FUNCTION_BLOCK "SSA_SIEMENS_MICROMASTER"	// FB 1813
TITLE = SIEMENS MICROMASTER
//COPYRIGHT:    (C) 2004  BUHLER AG, CH-9240 UZWIL, SWITZERLAND
//
//PRODUCT:      SSA
//
//TITLE:        SIEMENS MICROMASTER Frequency Inverter Profibus Communication
//
//--------------------------------------------------------------------------------
//
//IDENT:         AUTHOR:             DEPT:                            DATE:
//
//FB1813.2.0     M.Wedler            AEB41                            25-Okt-2007
//               2nd Release
//FB1811.1.0     A.Egli              CT3                              13-Jul-2007
//               1st Release
//
//--------------------------------------------------------------------------------
//
//PURPOSE: 
//
//MANUAL : 
//
//RESTRICTIONS: 
//
//--------------------------------------------------------------------------------
//
AUTHOR : MW
FAMILY : STD
VERSION : 0.0
VAR
  InValuePC : INT ;	//Aktuel value 1 in [0.01 %]
  InEnableRev : BOOL ;
  InEnableFwd : BOOL ;
  CmdFaultReset : BOOL ;
  OutRunningRev : BOOL ;	//Feedback for element motor
  OutRunningFwd : BOOL ;	//Feedback for element motor
  OutFault : BOOL ;	//Feedback for element motor
  MotorStStopped : BOOL ;	//Motor has come to a standstill after stopping time
  Spare : BOOL ;
  OutValuePC : INT ;	//Setpoint value 1 in [0.01 %]
  Input : STRUCT
   StateWord_1 : STRUCT 	//Statuswort MICROMASTER
    DREHZAHL_ABWEICHUNG_OK : BOOL ;	//0=Nicht im Toleranzband             1=Soll-Ist-Überwachung im Toleranzband
    FUEHRUNG : BOOL ;	//0=Fuehrung Lokal                    1=Fuehrung SPS
    VERGLEICHSWERT : BOOL ;	//0=Vergleichswert nicht erreicht     1=Vergleichswert erreicht/ueberschritten
    GRENZE_ERREICHT : BOOL ;	//0=I-, M- oder P-Grenze erreicht     1=I-, M- oder P-Grenze nicht erreicht
    HALTEBREMSE : BOOL ;	//0=Motor Haltebremse                 1=Steuern Haltebremse
    WARN_UEBERTEMP_MOTOR : BOOL ;	//0=Warnung nicht wirksam             1=Warnung Übertemperatur Motor wirksam
    DREH_RECHTS : BOOL ;	//0=Linkslauf                         1=Rechtslauf
    WARNUNG_UEBERTEMP_FU : BOOL ;	//0=Warnung thermische Überlast Umrichter 1=Keine Warnung wirksam
    EINSCHALTBEREIT : BOOL ;	//0=Nicht einschaltbereit             1=Einschaltbereit
    BETRIEBSBEREIT : BOOL ;	//0=Nicht betriebsbereit              1=Betriebsbereit
    BETRIEB_FREIGEGEBEN : BOOL ;	//0=Betrieb gesperrt   1=Betrieb freigegeben->Hochlauf auf anliegendem Sollwert
    STOERUNG : BOOL ;	//0=Keine Störung wirksam             1=Störung wirksam
    AUS_2 : BOOL ;	//0=Austrudeln aktiv (AUS2)           1=Kein AUS2 aktiv
    AUS_3 : BOOL ;	//0=Schnellhalt aktiv (AUS3)          1=Kein AUS3 aktiv
    EINSCHALTSPERRE : BOOL ;	//1=Einschaltsperre -> Wiedereinschalten durch AUS1 und anschließendes EIN
    WARNUNG : BOOL ;	//0=Keine Warnung wirksam             1=Warnung wirksam, Motor weiter im Betrieb
   END_STRUCT ;
   ActualValue01 : INT ;	//Hauptistwert / Prozessdaten PD2
   ActualValue02 : INT ;	//Prozessdaten PD3
   ActualValue03 : INT ;	//Prozessdaten PD4
   ActualValue04 : INT ;	//Prozessdaten PD5
   ActualValue05 : INT ;	//Prozessdaten PD6
  END_STRUCT ;
  Output : STRUCT
   ControlWord_1 : STRUCT 	//Steuerwort MICROMASTER
    TIPPEN_RECHTS : BOOL ;	//1=Tippen rechts
    TIPPEN_LINKS : BOOL ;	//1=Tippen links
    PZD_GUELTIG : BOOL ;	//0=Sollwerte ungueltig              1=Sollwerte gueltig
    DREHRICHTUNGSUMKEHR : BOOL ;	//Drehrichtungsumkehr: 0=Rechtsdrehfeld / 1=Linksdrehfeld
    CONTROL_WORD_BIT_12 : BOOL ;	//reserviert
    MOTOR_POTI_HIGH : BOOL ;	//1=Motorpotentiometer höher
    MOTOR_POTI_DOWN : BOOL ;	//1=Motorpotentiometer tiefer
    LOCAL : BOOL ;	//0=Fern-Steuerung aktiv             1=Vorort-Steuerung aktiv
    AUS1 : BOOL ;	//0=AUS1->Abbremsen an der Rücklauframpe   1=EIN
    AUS2 : BOOL ;	//0=Austrudeln (AUS2)                      1=kein Austrudeln
    AUS3 : BOOL ;	//0=Schnellhalt (AUS3)->Abbremsen an der Schnellhalt-Rampe  1=kein Schnellhalt
    BETRIEB_FREIGEBEN : BOOL ;	//0=Betrieb sperren        1=Betrieb freigeben->Hochlauf mit anliegendem Sollwert
    HOCHLAUF_SPERREN : BOOL ;	//0=Hochlaufgeber wird auf NULL gesetzt    1=Hochlaufgeber freigeben
    HOCHLAUF_STOPPEN : BOOL ;	//0=Hochlaufgeber einfrieren               1=Hochlaufgeber freigeben
    SOLLWERT_FREIGEBEN : BOOL ;	//0=Drehzahlsollwert wird auf NULL gesetzt 1=Drehzahlsollwert freigeben
    FEHLER_QUITTIEREN : BOOL ;	//Flanke 0 -> 1 = Fehler quittieren, quittiert alle aktuellen Störungen
   END_STRUCT ;
   SetpointValue01 : INT ;	//Hauptsollwert / Prozessdaten PD2
   SetpointValue02 : INT ;	//Prozessdaten PD3
   SetpointValue03 : INT ;	//Prozessdaten PD4
   SetpointValue04 : INT ;	//Prozessdaten PD5
   SetpointValue05 : INT ;	//Prozessdaten PD6
  END_STRUCT ;
  Par : STRUCT
   spare1 : INT ;
   spare2 : INT ;
   spare3 : INT ;
   ParMovidrive : BOOL ;
   ParSinamics : BOOL ;
   ParMicromaster : BOOL ;
   ParABB : BOOL ;
   ParNord : BOOL ;
   ParDanfoss : BOOL ;
   ParIOByteNo : INT ;
  END_STRUCT ;
END_VAR
VAR_TEMP
  tmpAddrDB : INT ;
  tmpAddrIO : DINT ;
  tmpAddrInputFU : DINT ;
  tmpAddrOutputFU : DINT ;
END_VAR
BEGIN
NETWORK
TITLE = Calculate Address of Inverter
      L     #Par.ParIOByteNo;
      SLD   3;
      T     #tmpAddrIO;
      L     P##Input;
      L     DW#16#FFFFFF;
      AD;
      TAR2;
      +D;
      T     #tmpAddrInputFU;
      L     P##Output;
      L     DW#16#FFFFFF;
      AD;
      TAR2;
      +D;
      T     #tmpAddrOutputFU;
NETWORK
TITLE = Prepare Commands Par.ParMicroMaster
      AN    #Par.ParNord;
      JC    MMJ0;
//Load Status Word
//      LAR1  #tmpAddrInputFU
//      L     DIW [AR1,P#0.0]             //Status Word
//      LAR1  P##MM_StateWord
//      T     LW [AR1,P#0.0]              // MM_StateWord
// prepare steuerword
      L     W#16#47E;	// Stop=AUS1
      A     #InEnableFwd;
      O     #InEnableRev;
      JCN   MMJ1;
      L     W#16#C7F;	// EIN + DREHRICHTUNGSUMKEHR
      A     #InEnableRev;
      JC    MMJ1;
      L     W#16#47F;	// Start=EIN
MMJ1: LAR1  #tmpAddrOutputFU;
      T     DIW [AR1,P#0.0];	// controlword 
//-----------------------------------------
// Fault Reset ins Steuerwort
      A     #CmdFaultReset;
      A     #Input.StateWord_1.STOERUNG;	// Fehler von FU
      JCN   MMR1;
      L     W#16#4FE;	// Reset ins Steuerwort
      LAR1  #tmpAddrOutputFU;
      T     DIW [AR1,P#0.0];	// controlword 
MMR1: NOP   0;
//- Feedback for motor
      A     #Input.StateWord_1.BETRIEB_FREIGEGEBEN;
      AN    #Input.StateWord_1.STOERUNG;
      A     #InEnableRev;
      =     #OutRunningRev;
      A     #Input.StateWord_1.BETRIEB_FREIGEGEBEN;
      AN    #Input.StateWord_1.STOERUNG;
      A     #InEnableFwd;
      =     #OutRunningFwd;
      A     #Input.StateWord_1.STOERUNG;
      =     #OutFault;
NETWORK
TITLE = Prepare setpoint value
//Motor nominal speed:
//4000H = 16384Dez = 100.0%
      L     #OutValuePC;
      ITD;
      DTR;
      L     1.638400e+00;
      *R;
      RND;
      T     #Output.SetpointValue01;
NETWORK
TITLE = Prepare actual value
//Motor nominal speed:
//4000H = 16384Dez = 100.0%
      L     #Input.ActualValue01;
      ITD;
      DTR;
      ABS;
      L     1.638400e+00;
      /R;
      RND;
      T     #InValuePC;
NETWORK
TITLE =
      A     #CmdFaultReset;
      R     #CmdFaultReset;
NETWORK
TITLE = Read Inputs of Inverter
      LAR1  #tmpAddrIO;
      L     PID [AR1,P#0.0];
      LAR1  #tmpAddrInputFU;
      T     DID [AR1,P#0.0];
      LAR1  #tmpAddrIO;
      L     PID [AR1,P#4.0];
      LAR1  #tmpAddrInputFU;
      T     DID [AR1,P#4.0];
      LAR1  #tmpAddrIO;
      L     PID [AR1,P#8.0];
      LAR1  #tmpAddrInputFU;
      T     DID [AR1,P#8.0];
NETWORK
TITLE = Write Outputs of Inverter
      LAR1  #tmpAddrOutputFU;
      L     DID [AR1,P#0.0];
      LAR1  #tmpAddrIO;
      T     PQD [AR1,P#0.0];
      LAR1  #tmpAddrOutputFU;
      L     DID [AR1,P#4.0];
      LAR1  #tmpAddrIO;
      T     PQD [AR1,P#4.0];
      LAR1  #tmpAddrOutputFU;
      L     DID [AR1,P#8.0];
      LAR1  #tmpAddrIO;
      T     PQD [AR1,P#8.0];
NETWORK
TITLE =
MMJ0: NOP   0;
      BE;
END_FUNCTION_BLOCK

FUNCTION_BLOCK "SSA_SIEMENS_SINAMICS"	// FB 1814
TITLE = SIEMENS SINAMICS
//COPYRIGHT:    (C) 2004  BUHLER AG, CH-9240 UZWIL, SWITZERLAND
//
//PRODUCT:      SSA
//
//TITLE:        SIEMENS SINAMICS Frequency Inverter Profibus Communication
//
//--------------------------------------------------------------------------------
//
//IDENT:         AUTHOR:             DEPT:                            DATE:
//
//FB1814.2.0     M.Wedler            AEB41                            25-Okt-2007
//               2nd Release
//FB1811.1.0     A.Egli              CT3                              13-Jul-2007
//               1st Release
//
//--------------------------------------------------------------------------------
//
//PURPOSE: 
//
//MANUAL : 
//
//RESTRICTIONS: 
//
//--------------------------------------------------------------------------------
//
AUTHOR : MW
FAMILY : STD
VERSION : 0.0
VAR
  InValuePC : INT ;	//Aktuel value 1 in [0.01 %]
  InEnableRev : BOOL ;
  InEnableFwd : BOOL ;
  CmdFaultReset : BOOL ;
  OutRunningRev : BOOL ;	//Feedback for element motor
  OutRunningFwd : BOOL ;	//Feedback for element motor
  OutFault : BOOL ;	//Feedback for element motor
  MotorStStopped : BOOL ;	//Motor has come to a standstill after stopping time
  Spare : BOOL ;
  OutValuePC : INT ;	//Setpoint value 1 in [0.01 %]
  Input : STRUCT
   StateWord_1 : STRUCT 	//Statuswort SINAMICS
    DREHZAHL_ABWEICHUNG_OK : BOOL ;	//0=Nicht im Toleranzband             1=Soll-Ist-Überwachung im Toleranzband
    FUEHRUNG : BOOL ;	//0=Fuehrung Lokal                    1=Fuehrung SPS
    VERGLEICHSWERT : BOOL ;	//0=Vergleichswert nicht erreicht     1=Vergleichswert erreicht/ueberschritten
    GRENZE_ERREICHT : BOOL ;	//0=I-, M- oder P-Grenze erreicht     1=I-, M- oder P-Grenze nicht erreicht
    STATE_WORD_BIT_12 : BOOL ;	//reserviert
    WARN_UEBERTEMP_MOTOR : BOOL ;	//0=Warnung nicht wirksam             1=Warnung Übertemperatur Motor wirksam
    DREH_RECHTS : BOOL ;	//0=Motor dreht nicht vorwärts        1=Motor dreht vorwärts
    WARNUNG_UEBERTEMP_FU : BOOL ;	//0=Warnung thermische Überlast Umrichter 1=Keine Warnung wirksam
    EINSCHALTBEREIT : BOOL ;	//0=Nicht einschaltbereit             1=Einschaltbereit
    BETRIEBSBEREIT : BOOL ;	//0=Nicht betriebsbereit              1=Betriebsbereit
    BETRIEB_FREIGEGEBEN : BOOL ;	//0=Betrieb gesperrt   1=Betrieb freigegeben->Hochlauf auf anliegendem Sollwert
    STOERUNG : BOOL ;	//0=Keine Störung wirksam             1=Störung wirksam
    AUS_2 : BOOL ;	//0=Austrudeln aktiv (AUS2)           1=Kein AUS2 aktiv
    AUS_3 : BOOL ;	//0=Schnellhalt aktiv (AUS3)          1=Kein AUS3 aktiv
    EINSCHALTSPERRE : BOOL ;	//1=Einschaltsperre -> Wiedereinschalten durch AUS1 und anschließendes EIN
    WARNUNG : BOOL ;	//0=Keine Warnung wirksam             1=Warnung wirksam
   END_STRUCT ;
   ActualValue01 : INT ;	//Hauptistwert / Prozessdaten PD2
   ActualValue02 : INT ;	//Prozessdaten PD3
   ActualValue03 : INT ;	//Prozessdaten PD4
   ActualValue04 : INT ;	//Prozessdaten PD5
   ActualValue05 : INT ;	//Prozessdaten PD6
  END_STRUCT ;
  Output : STRUCT
   ControlWord_1 : STRUCT 	//Steuerwort SINAMICS
    CONTROL_WORD_BIT_8 : BOOL ;	//reserviert
    CONTROL_WORD_BIT_9 : BOOL ;	//reserviert
    PZD_GUELTIG : BOOL ;	//Steuerworte, Sollwerte vom Profibus werden: 0=nicht ausgewertet / 1=ausgewertet
    DREHRICHTUNGSUMKEHR : BOOL ;	//Drehrichtungsumkehr: 0=Rechtsdrehfeld / 1=Linksdrehfeld
    CONTROL_WORD_BIT_12 : BOOL ;	//reserviert
    MOTOR_POTI_HIGH : BOOL ;	//1=Motorpotentiometer höher
    MOTOR_POTI_DOWN : BOOL ;	//1=Motorpotentiometer tiefer
    CONTROL_WORD_BIT_15 : BOOL ;	//reserviert
    AUS1 : BOOL ;	//0=AUS1->Abbremsen an der Rücklauframpe   1=EIN
    AUS2 : BOOL ;	//0=Austrudeln (AUS2)                      1=kein Austrudeln
    AUS3 : BOOL ;	//0=Schnellhalt (AUS3)->Abbremsen an der Schnellhalt-Rampe  1=kein Schnellhalt
    BETRIEB_FREIGEBEN : BOOL ;	//0=Betrieb sperren        1=Betrieb freigeben->Hochlauf mit anliegendem Sollwert
    HOCHLAUF_SPERREN : BOOL ;	//0=Hochlaufgeber wird auf NULL gesetzt    1=Hochlaufgeber freigeben
    HOCHLAUF_STOPPEN : BOOL ;	//0=Hochlaufgeber einfrieren               1=Hochlaufgeber wiederaufsetzen
    SOLLWERT_FREIGEBEN : BOOL ;	//0=Drehzahlsollwert wird auf NULL gesetzt 1=Drehzahlsollwert freigeben
    FEHLER_QUITTIEREN : BOOL ;	//Flanke 0 -> 1 = Fehler quittieren, quittiert alle aktuellen Störungen
   END_STRUCT ;
   SetpointValue01 : INT ;	//Hauptsollwert / Prozessdaten PD2
   SetpointValue02 : INT ;	//Prozessdaten PD3
   SetpointValue03 : INT ;	//Prozessdaten PD4
   SetpointValue04 : INT ;	//Prozessdaten PD5
   SetpointValue05 : INT ;	//Prozessdaten PD6
  END_STRUCT ;
  Par : STRUCT
   spare1 : INT ;
   spare2 : INT ;
   spare3 : INT ;
   ParMovidrive : BOOL ;
   ParSinamics : BOOL ;
   ParMicromaster : BOOL ;
   ParABB : BOOL ;
   ParNord : BOOL ;
   ParDanfoss : BOOL ;
   ParIOByteNo : INT ;
  END_STRUCT ;
END_VAR
VAR_TEMP
  tmpAddrDB : INT ;
  tmpAddrIO : DINT ;
  tmpAddrInputFU : DINT ;
  tmpAddrOutputFU : DINT ;
END_VAR
BEGIN
NETWORK
TITLE = Calculate Address of Inverter
      L     #Par.ParIOByteNo;
      SLD   3;
      T     #tmpAddrIO;
      L     P##Input;
      L     DW#16#FFFFFF;
      AD;
      TAR2;
      +D;
      T     #tmpAddrInputFU;
      L     P##Output;
      L     DW#16#FFFFFF;
      AD;
      TAR2;
      +D;
      T     #tmpAddrOutputFU;
NETWORK
TITLE = Prepare Commands Par.ParSinamics
      AN    #Par.ParSinamics;
      JC    SIJ0;
//Load Status Word
//      LAR1  #tmpAddrInputFU
//      L     DIW [AR1,P#0.0]             //Status Word
//      LAR1  P##SI_StateWord
//      T     LW [AR1,P#0.0]              // SI_StateWord
// prepare steuerword
      L     W#16#47E;	// Stop=AUS1
      A     #InEnableFwd;
      O     #InEnableRev;
      JCN   SIJ1;
      L     W#16#C7F;	// EIN + DREHRICHTUNGSUMKEHR
      A     #InEnableRev;
      JC    SIJ1;
      L     W#16#47F;	// Start=EIN
SIJ1: LAR1  #tmpAddrOutputFU;
      T     DIW [AR1,P#0.0];	// controlword 
//-----------------------------------------
// Fault Reset ins Steuerwort
      A     #CmdFaultReset;
      A     #Input.StateWord_1.STOERUNG;	// Fehler von FU
      JCN   SIR1;
      L     W#16#4FE;	// Reset ins Steuerwort
      LAR1  #tmpAddrOutputFU;
      T     DIW [AR1,P#0.0];	// controlword 
SIR1: NOP   0;
//- Feedback for motor
      A     #Input.StateWord_1.BETRIEB_FREIGEGEBEN;
      AN    #Input.StateWord_1.STOERUNG;
      A     #InEnableRev;
      =     #OutRunningRev;
      A     #Input.StateWord_1.BETRIEB_FREIGEGEBEN;
      AN    #Input.StateWord_1.STOERUNG;
      A     #InEnableFwd;
      =     #OutRunningFwd;
      A     #Input.StateWord_1.STOERUNG;
      =     #OutFault;
NETWORK
TITLE = Prepare setpoint value
//Motor nominal speed:
//4000H = 16384Dez = 100.0%
      L     #OutValuePC;
      ITD;
      DTR;
      L     1.638400e+00;
      *R;
      RND;
      T     #Output.SetpointValue01;
NETWORK
TITLE = Prepare actual value
//Motor nominal speed:
//4000H = 16384Dez = 100.0%
      L     #Input.ActualValue01;
      ITD;
      DTR;
      ABS;
      L     1.638400e+00;
      /R;
      RND;
      T     #InValuePC;
NETWORK
TITLE =
      A     #CmdFaultReset;
      R     #CmdFaultReset;
NETWORK
TITLE = Read Inputs of Inverter
      LAR1  #tmpAddrIO;
      L     PID [AR1,P#0.0];
      LAR1  #tmpAddrInputFU;
      T     DID [AR1,P#0.0];
      LAR1  #tmpAddrIO;
      L     PID [AR1,P#4.0];
      LAR1  #tmpAddrInputFU;
      T     DID [AR1,P#4.0];
      LAR1  #tmpAddrIO;
      L     PID [AR1,P#8.0];
      LAR1  #tmpAddrInputFU;
      T     DID [AR1,P#8.0];
NETWORK
TITLE = Write Outputs of Inverter
      LAR1  #tmpAddrOutputFU;
      L     DID [AR1,P#0.0];
      LAR1  #tmpAddrIO;
      T     PQD [AR1,P#0.0];
      LAR1  #tmpAddrOutputFU;
      L     DID [AR1,P#4.0];
      LAR1  #tmpAddrIO;
      T     PQD [AR1,P#4.0];
      LAR1  #tmpAddrOutputFU;
      L     DID [AR1,P#8.0];
      LAR1  #tmpAddrIO;
      T     PQD [AR1,P#8.0];
NETWORK
TITLE =
SIJ0: NOP   0;
      BE;
END_FUNCTION_BLOCK

FUNCTION_BLOCK "SSA_DANFOSS_VLT5000"	// FB 1815
TITLE = DANFOSS VLT5000
//COPYRIGHT:    (C) 2004  BUHLER AG, CH-9240 UZWIL, SWITZERLAND
//
//PRODUCT:      SSA
//
//TITLE:        DANFOSS VLT5000 Frequency Inverter Profibus Communication
//
//--------------------------------------------------------------------------------
//
//IDENT:         AUTHOR:             DEPT:                            DATE:
//
//FB1815.2.0     M.Wedler            AEB41                            29-Aug-2008
//               2nd Release
//FB1811.1.0     A.Egli              CT3                              13-Jul-2007
//               1st Release
//
//--------------------------------------------------------------------------------
//
//PURPOSE: 
//
//MANUAL : 
//
//RESTRICTIONS: 
//
//--------------------------------------------------------------------------------
//
AUTHOR : MW
FAMILY : STD
VERSION : 0.0
VAR
  InValuePC : INT ;	//Aktuel value 1 in [0.01 %]
  InEnableRev : BOOL ;
  InEnableFwd : BOOL ;
  CmdFaultReset : BOOL ;
  OutRunningRev : BOOL ;	//Feedback for element motor
  OutRunningFwd : BOOL ;	//Feedback for element motor
  OutFault : BOOL ;	//Feedback for element motor
  MotorStStopped : BOOL ;	//Motor has come to a standstill after stopping time
  Spare : BOOL ;
  OutValuePC : INT ;	//Setpoint value 1 in [0.01 %]
  Input : STRUCT
   StateWord_1 : STRUCT 	//Statuswort VLT 5000
    _ACT_VALUE : BOOL ;	//0=Set <> act                                  1=set==act value
    _MODE : BOOL ;	//0=local mode                                  1=Profibus mode
    _FREQUENZ_OK : BOOL ;	//0=Frequenz out of limits                      1=act Frequenz ok
    _RUNNING : BOOL ;	//0=Motor stopped                               1=motor running
    _OVERLOAD : BOOL ;	//0=no overload                                 1=FU overload
    _FU_VOLTAGE_OK : BOOL ;	//0=FU Voltage ok                               1=FU voltage out of limits
    _FU_MOMENT_OK : BOOL ;	//0=FU moment ok                                1=FU moment out of limits
    _FU_THERMIC_OVERLOAD : BOOL ;	//0=FU thermic overload ok                      1=FU thermic overload
    _CONTROL_SYSTEM : BOOL ;	//0=Control System fault                        1=control System OK
    _VLT_OK : BOOL ;	//0=VLT not ok (incl.power)                     1=VLT ok (incl.power)
    _FREILAUF : BOOL ;	//0=Freilauf, FU hat abgeschaltet               1=kein Freilauf = ok
    _FAULT : BOOL ;	//0=No Fault                                    1=Fault, Reset required
    _RESERVE0_4 : BOOL ;	//not used
    _RESERVE0_5 : BOOL ;	//not used
    _RESERVE0_6 : BOOL ;	//not used
    _WARNUNG : BOOL ;	//0=ok                                          1=warning FU
   END_STRUCT ;
   ActualValue01 : INT ;	//Hauptistwert / Prozessdaten PD2
   ActualValue02 : INT ;	//Prozessdaten PD3
   ActualValue03 : INT ;	//Prozessdaten PD4
   ActualValue04 : INT ;	//Prozessdaten PD5
   ActualValue05 : INT ;	//Prozessdaten PD6
   STAT0 : BOOL ;
  END_STRUCT ;
  Output : STRUCT
   ControlWord_1 : STRUCT 	//Steuerwort VLT 5000
    _BETRIEBSART : BOOL ;	//0=normalbetrieb                    1=Jog (motor läuft mit Festdrehzahl)
    _RAMPE1_2 : BOOL ;	//0=Rampe 1 aktiv                    0=Rampe 2 aktiv
    _PROFIBUS : BOOL ;	//1=Daten über Profibus !!!          0=lokalbetrieb
    _RELAIS1 : BOOL ;	//0=Relais1 nicht aktiv              1=Relais1 aktiv
    _RELAIS4 : BOOL ;	//0=Relais4 nicht aktiv              1=Relais4 aktiv
    _PARAMETERSATZ1 : BOOL ;	//0-3 = Selection Parametersatz 1-4
    _PARAMETERSATZ4 : BOOL ;	//0-3 = Selection Parametersatz 1-4
    _NORMALLAUF : BOOL ;	//0=Normallauf                       1=Reversierung
    _AUS1 : BOOL ;	//0-3 = Selection Parameter 215-218 fix set Value
    _AUS2 : BOOL ;	//0-3 = Selection Parameter 215-218 fix set Value
    _RAMPE : BOOL ;	//1=Rampe                            0=Bremsen
    _NORMALBETRIEB : BOOL ;	//1=normalbetrieb                    0=Stopp mit Freilauf
    _SCHNELLSTOPP : BOOL ;	//1=Rampe                            0=SchnellStopp mit Rampe
    _SET1 : BOOL ;	//1=Rampe möglich (muss immer 1 sein!)
    _START : BOOL ;	//1=Start                            0=normaler Rampenstopp
    _RESET : BOOL ;	//1-Flanke =Reset nach Abschaltung   0=keine Funktion
   END_STRUCT ;
   SetpointValue01 : INT ;	//Hauptsollwert / Prozessdaten PD2
   SetpointValue02 : INT ;	//Prozessdaten PD3
   SetpointValue03 : INT ;	//Prozessdaten PD4
   SetpointValue04 : INT ;	//Prozessdaten PD5
   SetpointValue05 : INT ;	//Prozessdaten PD6
   STAT34 : BOOL ;
  END_STRUCT ;
  Par : STRUCT
   spare1 : INT ;
   spare2 : INT ;
   spare3 : INT ;
   ParMovidrive : BOOL ;
   ParSinamics : BOOL ;
   ParMicromaster : BOOL ;
   ParABB : BOOL ;
   ParNord : BOOL ;
   ParDanfoss : BOOL ;
   ParIOByteNo : INT ;
  END_STRUCT ;
END_VAR
VAR_TEMP
  tmpAddrDB : INT ;
  tmpAddrIO : DINT ;
  tmpAddrInputFU : DINT ;
  tmpAddrOutputFU : DINT ;
END_VAR
BEGIN
NETWORK
TITLE = Calculate Address of Inverter
      L     #Par.ParIOByteNo;	//Laden FU Adresse
      SLD   3;	//Wandeln in Pointer Format
      T     #tmpAddrIO;	//Pointer Speichern
      L     P##Input;	//Adresse Laden von Zustandsworten
      L     DW#16#FFFFFF;	//Bereinigen von DW 
      AD;	//UND - Doppelwort
      TAR2;	//Transfert ADDR2 in AKKU1
      +D;	//Adition Doppelwort
      T     #tmpAddrInputFU;
      L     P##Output;
      L     DW#16#FFFFFF;
      AD;
      TAR2;
      +D;
      T     #tmpAddrOutputFU;
NETWORK
TITLE = Prepare Commands Par.ParDanfoss
//! Test commands for VLT FC100 !
      AN    #Par.ParDanfoss;
      JC    DAJ0;
//Load Status Word
//      LAR1  #tmpAddrInputFU
//      L     DIW [AR1,P#0.0]             //Status Word
//      LAR1  P##DANFOSS_StateWord
//      T     LW [AR1,P#0.0]              // DANFOSS_StateWord
// prepare steuerword
      L     W#16#43E;	// Stop FC  //[2.0]
      A     #InEnableFwd;	//[2.0]
      O     #InEnableRev;	//[2.0]
      JCN   DAJ1;	//[2.0]
      L     W#16#847F;	// Start FC revers  //[2.0]
      A     #InEnableRev;	//[2.0]
      JC    DAJ1;	//[2.0]
      L     W#16#47F;	// Start FC   //[2.0]
DAJ1: LAR1  #tmpAddrOutputFU;
      T     DIW [AR1,P#0.0];	// controlword 
//-----------------------------------------
// Fault Reset ins Steuerwort
// VLT5000 - Not tested                  //[2.0]                
//      U     #Input.StateWord_1._OVERLOAD    // Fehler von FU
//      O     #Input.StateWord_1._FU_THERMIC_OVERLOAD    // Fehler von FU
// FC100 - Tested by UAN01         //[2.0]
      A     #Input.StateWord_1._FAULT;	// FC100    //[2.0]
      A     #CmdFaultReset;
      JCN   DAR1;
      L     W#16#48E;	// Reset ins Steuerwort
      LAR1  #tmpAddrOutputFU;
      T     DIW [AR1,P#0.0];	// controlword 
DAR1: NOP   0;
//- Feedback for motor
// VLT5000 - Not tested      //[2.0]
//      U     #Input.StateWord_1._RUNNING // VLT5000   //[2.0]
//      UN    #Input.StateWord_1._OVERLOAD    // Fehler von FU    //[2.0]
//      UN    #Input.StateWord_1._FU_THERMIC_OVERLOAD    // Fehler von FU  //[2.0]
// FC100 - Tested by UAN01                  //[2.0]
      A     #Input.StateWord_1._FREQUENZ_OK;	// FC100   //[2.0]
      A     #Input.StateWord_1._RUNNING;	// FC100  //[2.0]
      AN    #Input.StateWord_1._FAULT;	// FC100  //[2.0]
      A     #InEnableRev;	//[2.0]
      =     #OutRunningRev;	//[2.0]
// VLT5000 - Not tested                                //[2.0]
//      U     #Input.StateWord_1._RUNNING // VLT5000    //[2.0]
//      UN    #Input.StateWord_1._OVERLOAD    // Fehler von FU  //[2.0]
//      UN    #Input.StateWord_1._FU_THERMIC_OVERLOAD    // Fehler von FU  //[2.0]
// FC100 - Tested by UAN01                //[2.0]
      A     #Input.StateWord_1._FREQUENZ_OK;	// FC100   //[2.0]
      A     #Input.StateWord_1._RUNNING;	// FC100     //[2.0]
      AN    #Input.StateWord_1._FAULT;	// FC100     //[2.0]
      A     #InEnableFwd;	//[2.0]
      =     #OutRunningFwd;	//[2.0]
// VLT5000 - Not tested                  //[2.0]                
//      U     #Input.StateWord_1._OVERLOAD    // Fehler von FU   //[2.0]
//      O     #Input.StateWord_1._FU_THERMIC_OVERLOAD    // Fehler von FU    //[2.0]
// FC100 - Tested by UAN01         //[2.0]
      A     #Input.StateWord_1._FAULT;	// FC100    //[2.0]
      =     #OutFault;	//[2.0]
NETWORK
TITLE = Prepare setpoint value
//Motor nominal speed:
//4000H = 16384Dez = 100.0%
      L     #OutValuePC;
      ITD;
      DTR;
      L     1.638400e+00;
      *R;
      RND;
      T     #Output.SetpointValue01;
NETWORK
TITLE = Prepare actual value
//Motor nominal speed:
//4000H = 16384Dez = 100.0%
      L     #Input.ActualValue01;
      ITD;
      DTR;
      ABS;
      L     1.638400e+00;
      /R;
      RND;
      T     #InValuePC;
NETWORK
TITLE =
      A     #CmdFaultReset;
      R     #CmdFaultReset;
NETWORK
TITLE = Read Inputs of Inverter
      LAR1  #tmpAddrIO;
      L     PID [AR1,P#0.0];
      LAR1  #tmpAddrInputFU;
      T     DID [AR1,P#0.0];
      LAR1  #tmpAddrIO;
      L     PID [AR1,P#4.0];
      LAR1  #tmpAddrInputFU;
      T     DID [AR1,P#4.0];
      LAR1  #tmpAddrIO;
      L     PID [AR1,P#8.0];
      LAR1  #tmpAddrInputFU;
      T     DID [AR1,P#8.0];
NETWORK
TITLE = Write Outputs of Inverter
      LAR1  #tmpAddrOutputFU;
      L     DID [AR1,P#0.0];
      LAR1  #tmpAddrIO;
      T     PQD [AR1,P#0.0];
      LAR1  #tmpAddrOutputFU;
      L     DID [AR1,P#4.0];
      LAR1  #tmpAddrIO;
      T     PQD [AR1,P#4.0];
      LAR1  #tmpAddrOutputFU;
      L     DID [AR1,P#8.0];
      LAR1  #tmpAddrIO;
      T     PQD [AR1,P#8.0];
NETWORK
TITLE =
DAJ0: NOP   0;
      BE;
END_FUNCTION_BLOCK

FUNCTION_BLOCK "SSA_ABB"	// FB 1816
TITLE = ABB ACS800
//COPYRIGHT:    (C) 2004  BUHLER AG, CH-9240 UZWIL, SWITZERLAND
//
//PRODUCT:      SSA
//
//TITLE:        ABB ACS800 Frequency Inverter Profibus Communication
//
//--------------------------------------------------------------------------------
//
//IDENT:         AUTHOR:             DEPT:                            DATE:
//
//FB1816.2.1     M.Wedler            AEB41                            07-Nov-2008
//               Assignation of MotorStStopped internal 
//FB1816.2.0     M.Wedler            AEB41                            25-Okt-2007
//               2nd Release
//FB1811.1.0     A.Egli              CT3                              13-Jul-2007
//               1st Release
//
//--------------------------------------------------------------------------------
//
//PURPOSE: 
//
//MANUAL : 
//
//RESTRICTIONS: 
//
//--------------------------------------------------------------------------------
//
AUTHOR : MW
FAMILY : STD
VERSION : 0.0
VAR
  InValuePC : INT ;	//Aktuel value 1 in [0.01 %]
  InEnableRev : BOOL ;
  InEnableFwd : BOOL ;
  CmdFaultReset : BOOL ;
  OutRunningRev : BOOL ;	//Feedback for element motor
  OutRunningFwd : BOOL ;	//Feedback for element motor
  OutFault : BOOL ;	//Feedback for element motor
  MotorStStopped : BOOL ;	//Motor has come to a standstill after stopping time
  Spare : BOOL ;
  OutValuePC : INT ;	//Setpoint value 1 in [0.01 %]
  Input : STRUCT
   StateWord_1 : STRUCT 	//State Word ABB
    AT_SETPOINT : BOOL ;	//0=Actual value differs from reference valu; 1=Actual value equals reference val
    REMOTE : BOOL ;	//0=LOCAL                         1=REMOTE
    ABOVE_LIMIT : BOOL ;	//0=within supervision limit      1=equals or is greater than supervision limit
    STATE_WORD_BIT_11 : BOOL ;	//Drive-specific
    STATE_WORD_BIT_12 : BOOL ;	//Drive-specific
    STATE_WORD_BIT_13 : BOOL ;	//Drive-specific
    STATE_WORD_BIT_14 : BOOL ;	//Drive-specific
    STATE_WORD_BIT_15 : BOOL ;	//Drive-specific
    RDY_ON : BOOL ;	//0=NOT READY TO SWITCH ON        1=READY TO SWITCH ON
    RDY_RUN : BOOL ;	//0=OFF1 ACTIVE                   1=READY TO OPERATE
    RDY_REF : BOOL ;	//0=DISABLE OPERATION             1=ENABLE OPERATION
    TRIPPED : BOOL ;	//0=No fault                      1=FAULT
    OFF_2_STA : BOOL ;	//0=OFF2 ACTIVE                   1=OFF2 inactive
    OFF_3_STA : BOOL ;	//0=OFF3 ACTIVE                   1=OFF3 inactive
    SWC_ON_INHIB : BOOL ;	//0=SWITCH-ON INHIBIT NOT ACTIVE  1=SWITCH-ON INHIBIT ACTIVE
    ALARM : BOOL ;	//0=No Warning/Alarm              1=Warning/Alarm
   END_STRUCT ;
   ActualValue01 : INT ;	//ACTUAL VALUE / the actual speed (0-4000h) corresponds to 0-motor nominal speed
   ActualValue02 : INT ;	//Process Data PZD3
   ActualValue03 : INT ;	//Process Data PZD4
   ActualValue04 : INT ;	//Process Data PZD5
   ActualValue05 : INT ;	//Process Data PZD6
  END_STRUCT ;
  Output : STRUCT
   ControlWord_1 : STRUCT 	//Control Word ABB
    INCHING_1 : BOOL ;	//Inching 1.
    INCHING_2 : BOOL ;	//Inching 2.
    REMOTE_CMD : BOOL ;	//0=Retain last Control Word and Reference        1=Fieldbus control enabled
    CONTROL_WORD_BIT_11 : BOOL ;	//Drive-specific
    CONTROL_WORD_BIT_12 : BOOL ;	//Drive-specific
    CONTROL_WORD_BIT_13 : BOOL ;	//Drive-specific
    CONTROL_WORD_BIT_14 : BOOL ;	//Drive-specific
    CONTROL_WORD_BIT_15 : BOOL ;	//Drive-specific
    OFF1 : BOOL ;	//0=Emergency OFF-stop by the selected deceleration 1=Proceed to READY TO OPERATE
    OFF2 : BOOL ;	//0=Emergency OFF-coast to stop              1=Continue operation (OFF2 inactive)
    OFF3 : BOOL ;	//0=Emergency stop-stop according to fastest possible deceleration mode
    OPERATION_ENABLE : BOOL ;	//0=Inhibit operation                             1=Proceed to ENABLE OPERATION
    RAMP_OUT_ZERO : BOOL ;	//0=Stop according to selected stop type          1=Normal operation
    RAMP_HOLD : BOOL ;	//0=Halt ramping                                  1=Normal operation
    RAMP_IN_ZERO : BOOL ;	//0=Force Ramp Function Generator input to zero   1=Normal operation
    RESET : BOOL ;	//1=Fault reset if an active fault exists
   END_STRUCT ;
   SetpointValue01 : INT ;	//REFERENCE / the speed reference (0-4000h) corresponds to 0-motor nominal speed
   SetpointValue02 : INT ;	//Process Data PZD3
   SetpointValue03 : INT ;	//Process Data PZD4
   SetpointValue04 : INT ;	//Process Data PZD5
   SetpointValue05 : INT ;	//Process Data PZD6
  END_STRUCT ;
  Par : STRUCT
   spare1 : INT ;
   spare2 : INT ;
   spare3 : INT ;
   ParMovidrive : BOOL ;
   ParSinamics : BOOL ;
   ParMicromaster : BOOL ;
   ParABB : BOOL ;
   ParNord : BOOL ;
   ParDanfoss : BOOL ;
   ParIOByteNo : INT ;
  END_STRUCT ;
END_VAR
VAR_TEMP
  tmpAddrDB : INT ;
  tmpAddrIO : DINT ;
  tmpAddrInputFU : DINT ;
  tmpAddrOutputFU : DINT ;
END_VAR
BEGIN
NETWORK
TITLE = Calculate Address of Inverter
      L     #Par.ParIOByteNo;
      SLD   3;
      T     #tmpAddrIO;
      L     P##Input;
      L     DW#16#FFFFFF;
      AD;
      TAR2;
      +D;
      T     #tmpAddrInputFU;
      L     P##Output;
      L     DW#16#FFFFFF;
      AD;
      TAR2;
      +D;
      T     #tmpAddrOutputFU;
NETWORK
TITLE = Prepare Commands Par.ParABB
//Erklärung für Unbeteiligte:
//
//1. Wenn FU ohne Rampe gestoppt wird (Austrudeln), dann
//a) L  W#16#477  // DISABLE OPERATION (Austrudeln)
//und wenn Motor steht (Drehzahl = ca. 0 rpm)   
//b) L  W#16#476  // DISABLE OPERATION + Emergency OFF-stop by the selected 
//deceleration (Not-Halt, anhalten mit der eingestellten Verzögerungsrampe)
//
//2. Wenn FU mit Rampe gestoppt wird (Stopprampe), dann
//a) L  W#16#47E  // Emergency OFF-stop by the selected deceleration 
//(Stopp mit Rampe)
//
      AN    #Par.ParABB;
      JC    ABJ0;
//Load Status Word
//      LAR1  #tmpAddrInputFU
//      L     DIW [AR1,P#0.0]             // Status Word
//      LAR1  P##ABB_StateWord
//      T     LW [AR1,P#0.0]              // ABB_StateWord
// prepare steuerword
// DISABLE OPERATION + Emergency OFF-stop by the selected deceleration  
// (Not-Halt, anhalten mit der eingestellten Verzögerungsrampe)
      L     W#16#476;
      AN    #InEnableFwd;
      AN    #InEnableRev;
      A     #MotorStStopped;	// Standstill of motor
      O     #Input.StateWord_1.TRIPPED;	// FAULT (Fehler)
      JC    ABJ1;
// Stopp without ramp 
      L     W#16#477;	// DISABLE OPERATION (Austrudeln)
// or stopp with ramp
// Emergency OFF-stop by the selected deceleration (Stopp mit Rampe)
//      L     W#16#47E     // DISABLE OPERATION + Emergency OFF             
      A     #InEnableFwd;
      O     #InEnableRev;
      JCN   ABJ1;
      L     W#16#47F;	// Start=EIN
ABJ1: LAR1  #tmpAddrOutputFU;
      T     DIW [AR1,P#0.0];	// controlword 
//-----------------------------------------
// Fault Reset ins Steuerwort
      A     #CmdFaultReset;
      A     #Input.StateWord_1.TRIPPED;	// FAULT (Fehler)
      JCN   ABR1;
      L     W#16#4FE;	// Reset ins Steuerwort
      LAR1  #tmpAddrOutputFU;
      T     DIW [AR1,P#0.0];	// controlword 
ABR1: NOP   0;
//- Feedback for motor
      A     #Input.StateWord_1.RDY_REF;
      AN    #Input.StateWord_1.TRIPPED;
      A     #InEnableRev;
      =     #OutRunningRev;
      A     #Input.StateWord_1.RDY_REF;
      AN    #Input.StateWord_1.TRIPPED;
      A     #InEnableFwd;
      =     #OutRunningFwd;
      A     #Input.StateWord_1.TRIPPED;
      =     #OutFault;
NETWORK
TITLE = Prepare setpoint value
//Motor nominal speed:
//+20000Dez = +100.0%
//-20000Dez = -100.0%
      L     #OutValuePC;
      ITD;
      DTR;
      L     2.000000e+00;
      *R;
      RND;
      A     #InEnableRev;
      JCN   tsp;
      NEGD;
tsp:  T     #Output.SetpointValue01;
NETWORK
TITLE = Prepare actual value
//Motor nominal speed:
//+20000Dez = +100.0%
//-20000Dez = -100.0%
      L     #Input.ActualValue01;
      ITD;
      DTR;
      ABS;
      L     2.000000e+00;
      /R;
      RND;
      T     #InValuePC;
//-Assignation of MotorStStopped internal      [2.1]
      L     #Input.ActualValue01;
      L     200;	// 200Dez = 1.0%Fn
      >I;
      A     #Input.StateWord_1.RDY_REF;
      JCN   MSta;
      CLR;
      =     #MotorStStopped;	// Standstill of motor
MSta: NOP   0;
      L     #Input.ActualValue01;
      L     200;	// 200Dez = 1.0%Fn
      <I;
      JCN   MSto;
      SET;
      =     #MotorStStopped;	// Standstill of motor
MSto: NOP   0;
NETWORK
TITLE =
      A     #CmdFaultReset;
      R     #CmdFaultReset;
NETWORK
TITLE = Read Inputs of Inverter
      LAR1  #tmpAddrIO;
      L     PID [AR1,P#0.0];
      LAR1  #tmpAddrInputFU;
      T     DID [AR1,P#0.0];
      LAR1  #tmpAddrIO;
      L     PID [AR1,P#4.0];
      LAR1  #tmpAddrInputFU;
      T     DID [AR1,P#4.0];
      LAR1  #tmpAddrIO;
      L     PID [AR1,P#8.0];
      LAR1  #tmpAddrInputFU;
      T     DID [AR1,P#8.0];
NETWORK
TITLE = Write Outputs of Inverter
      LAR1  #tmpAddrOutputFU;
      L     DID [AR1,P#0.0];
      LAR1  #tmpAddrIO;
      T     PQD [AR1,P#0.0];
      LAR1  #tmpAddrOutputFU;
      L     DID [AR1,P#4.0];
      LAR1  #tmpAddrIO;
      T     PQD [AR1,P#4.0];
      LAR1  #tmpAddrOutputFU;
      L     DID [AR1,P#8.0];
      LAR1  #tmpAddrIO;
      T     PQD [AR1,P#8.0];
NETWORK
TITLE =
ABJ0: NOP   0;
      BE;
END_FUNCTION_BLOCK

FUNCTION_BLOCK "SSA_NORD"	// FB 1817
TITLE = NORDAC
//COPYRIGHT:    (C) 2004  BUHLER AG, CH-9240 UZWIL, SWITZERLAND
//
//PRODUCT:      SSA
//
//TITLE:        NORDAC Frequency Inverter Profibus Communication
//
//--------------------------------------------------------------------------------
//
//IDENT:         AUTHOR:             DEPT:                            DATE:
//
//FB1817.2.0     M.Wedler            AEB41                            25-Okt-2007
//               2nd Release
//FB1811.1.0     A.Egli              CT3                              13-Jul-2007
//               1st Release
//
//--------------------------------------------------------------------------------
//
//PURPOSE: 
//
//MANUAL : 
//
//RESTRICTIONS: 
//
//--------------------------------------------------------------------------------
//
AUTHOR : MW
FAMILY : STD
VERSION : 0.0
VAR
  InValuePC : INT ;	//Aktuel value 1 in [0.01 %]
  InEnableRev : BOOL ;
  InEnableFwd : BOOL ;
  CmdFaultReset : BOOL ;
  OutRunningRev : BOOL ;	//Feedback for element motor
  OutRunningFwd : BOOL ;	//Feedback for element motor
  OutFault : BOOL ;	//Feedback for element motor
  MotorStStopped : BOOL ;	//Motor has come to a standstill after stopping time
  Spare : BOOL ;
  OutValuePC : INT ;	//Setpoint value 1 in [0.01 %]
  Input : STRUCT
   StateWord_1 : STRUCT 	//State Word NORDAC
    ACTUAL_VALUE_OK : BOOL ;	//0=Actual value doesn't match setpoint  1=Actual value matches required setpoint
    GUIDANCE : BOOL ;	//0=Local guidance                       1=Guidance requested
    ACTUAL_MFR1_VALUE : BOOL ;	//0=Actual MFR 1 value below reference value    1=MFR 1 value has been equalled
    ROTAT_DIRECTION_RIGHT : BOOL ;	//1=Inverter output voltage is turning right
    ROTAT_DIRECTION_LEFT : BOOL ;	//1=Inverter output voltage is turning left
    ACTUAL_MFR4_VALUE : BOOL ;	//Only with SK 700E/750E with posicon extension Status MFR 4
    PARAMETER_SET_0 : BOOL ;	//00=Parameter set 1 01=Parameter set 2 10=Parameter set 3 11=Parameter set 4
    PARAMETER_SET_1 : BOOL ;	//00=Parameter set 1 01=Parameter set 2 10=Parameter set 3 11=Parameter set 4
    READY_TO_START : BOOL ;	//0=Not ready to start                   1=Ready to start
    READY_FOR_OPERATION : BOOL ;	//0=Not ready for operation              1=Ready for operation
    OPERATION_ENABLED : BOOL ;	//0=Operation disabled                   1=Operation enabled
    FAULT : BOOL ;	//0=No fault                             1=Fault
    OFF2 : BOOL ;	//0=OFF2 command applied                 1=no OFF2
    OFF3 : BOOL ;	//0=OFF3 command applied                 1=no OFF3
    STARTING_DISABLED : BOOL ;	//0=Starting not disabled                1=Starting disabled
    WARNING : BOOL ;	//0=No warning                           1=Warning
   END_STRUCT ;
   ActualValue01 : INT ;	//Actual frequency. 4000H = 100%, C000H = -100% of maximum frequency
   ActualValue02 : INT ;	//Process Data PZD3
   ActualValue03 : INT ;	//Process Data PZD4
   ActualValue04 : INT ;	//Not used
   ActualValue05 : INT ;	//Not used
  END_STRUCT ;
  Output : STRUCT
   ControlWord_1 : STRUCT 	//Control Word NORDAC
    RESERVED_8 : BOOL ;	//Reserved
    RESERVED_9 : BOOL ;	//Reserved
    PZD_VALID : BOOL ;	//0=The transmitted process data is invalid  1=Valid process data transferred
    ROTAT_DIRECTION_RIGHT : BOOL ;	//1=Rotational direction right ON
    ROTAT_DIRECTION_LEFT : BOOL ;	//1=Rotational direction left ON
    RESERVED_13 : BOOL ;	//Reserved
    SWITCH_PARAMETER_SET_0 : BOOL ;	//00=Parameter set 1 01=Parameter set 2 10=Parameter set 3 11=Parameter set 4
    SWITCH_PARAMETER_SET_1 : BOOL ;	//00=Parameter set 1 01=Parameter set 2 10=Parameter set 3 11=Parameter set 4
    OFF1 : BOOL ;	//0=Reverse with the brake ramp              1=Ready for operation
    OFF2 : BOOL ;	//0=Inverter output voltage is switched off  1=OFF 2 is cancelled
    OFF3 : BOOL ;	//0=Quick stop with programmed quick stop time  1=OFF 3 is cancelled
    ENABLE_OPERATION : BOOL ;	//0=Disable operation                        1=Enable operation
    LOCK_RAMP_GENERATOR : BOOL ;	//0=Ramp generator is set to zero            1=Enable ramp generator
    STOP_RAMP_GENERATOR : BOOL ;	//0=The setpoint currently provided by the ramp generator is "frozen"
    DISABLE_SETPOINT : BOOL ;	//0=Selected setpoint value is set to zero on the ramp generator
    ACKNOWLEDGE : BOOL ;	//0->1=Acknowledgement of faults which are no longer active
   END_STRUCT ;
   SetpointValue01 : INT ;	//Setpoint frequency. 4000H = 100%, C000H = -100% of maximum frequency
   SetpointValue02 : INT ;	//Process Data PZD3
   SetpointValue03 : INT ;	//Process Data PZD4
   SetpointValue04 : INT ;	//Not used
   SetpointValue05 : INT ;	//Not used
  END_STRUCT ;
  Par : STRUCT
   spare1 : INT ;
   spare2 : INT ;
   spare3 : INT ;
   ParMovidrive : BOOL ;
   ParSinamics : BOOL ;
   ParMicromaster : BOOL ;
   ParABB : BOOL ;
   ParNord : BOOL ;
   ParDanfoss : BOOL ;
   ParIOByteNo : INT ;
  END_STRUCT ;
END_VAR
VAR_TEMP
  tmpAddrDB : INT ;
  tmpAddrIO : DINT ;
  tmpAddrInputFU : DINT ;
  tmpAddrOutputFU : DINT ;
END_VAR
BEGIN
NETWORK
TITLE = Calculate Address of Inverter
      L     #Par.ParIOByteNo;
      SLD   3;
      T     #tmpAddrIO;
      L     P##Input;
      L     DW#16#FFFFFF;
      AD;
      TAR2;
      +D;
      T     #tmpAddrInputFU;
      L     P##Output;
      L     DW#16#FFFFFF;
      AD;
      TAR2;
      +D;
      T     #tmpAddrOutputFU;
NETWORK
TITLE = Prepare Commands Par.ParNord
      AN    #Par.ParNord;
      JC    NOJ0;
//Load Status Word
//      LAR1  #tmpAddrInputFU
//      L     DIW [AR1,P#0.0]             //Status Word
//      LAR1  P##NORD_StateWord
//      T     LW [AR1,P#0.0]              // NORD_StateWord
// prepare steuerword
      L     W#16#47E;	// Stopp=OFF1
      A     #InEnableFwd;
      O     #InEnableRev;
      JCN   NOJ1;
      L     W#16#147F;	// Start direction left 
      A     #InEnableRev;
      JC    NOJ1;
      L     W#16#C7F;	// Start direction right
NOJ1: LAR1  #tmpAddrOutputFU;
      T     DIW [AR1,P#0.0];	// controlword 
//-----------------------------------------
// Fault Reset ins Steuerwort
      A     #CmdFaultReset;
      A     #Input.StateWord_1.FAULT;	// Fehler von FU
      JCN   NOR1;
      L     W#16#4FE;	// OFF1 + ACKNOWLEDGE
      LAR1  #tmpAddrOutputFU;
      T     DIW [AR1,P#0.0];	// controlword 
NOR1: NOP   0;
//- Feedback for motor
      A     #Input.StateWord_1.OPERATION_ENABLED;
      AN    #Input.StateWord_1.FAULT;
      A     #InEnableRev;
      =     #OutRunningRev;
      A     #Input.StateWord_1.OPERATION_ENABLED;
      AN    #Input.StateWord_1.FAULT;
      A     #InEnableFwd;
      =     #OutRunningFwd;
      A     #Input.StateWord_1.FAULT;
      =     #OutFault;
NETWORK
TITLE = Prepare setpoint value
//Motor nominal speed:
//4000H = 16384Dez = 100.0%
      L     #OutValuePC;
      ITD;
      DTR;
      L     1.638400e+00;
      *R;
      RND;
      T     #Output.SetpointValue01;
NETWORK
TITLE = Prepare actual value
//Motor nominal speed:
//4000H = 16384Dez = 100.0%
      L     #Input.ActualValue01;
      ITD;
      DTR;
      ABS;
      L     1.638400e+00;
      /R;
      RND;
      T     #InValuePC;
NETWORK
TITLE =
      A     #CmdFaultReset;
      R     #CmdFaultReset;
NETWORK
TITLE = Read Inputs of Inverter
      LAR1  #tmpAddrIO;
      L     PID [AR1,P#0.0];
      LAR1  #tmpAddrInputFU;
      T     DID [AR1,P#0.0];
      LAR1  #tmpAddrIO;
      L     PID [AR1,P#4.0];
      LAR1  #tmpAddrInputFU;
      T     DID [AR1,P#4.0];
      LAR1  #tmpAddrIO;
      L     PID [AR1,P#8.0];
      LAR1  #tmpAddrInputFU;
      T     DID [AR1,P#8.0];
NETWORK
TITLE = Write Outputs of Inverter
      LAR1  #tmpAddrOutputFU;
      L     DID [AR1,P#0.0];
      LAR1  #tmpAddrIO;
      T     PQD [AR1,P#0.0];
      LAR1  #tmpAddrOutputFU;
      L     DID [AR1,P#4.0];
      LAR1  #tmpAddrIO;
      T     PQD [AR1,P#4.0];
      LAR1  #tmpAddrOutputFU;
      L     DID [AR1,P#8.0];
      LAR1  #tmpAddrIO;
      T     PQD [AR1,P#8.0];
NETWORK
TITLE =
NOJ0: NOP   0;
      BE;
END_FUNCTION_BLOCK

FUNCTION_BLOCK "SSA_SEW_MOVITRAC"	// FB 1818
TITLE = SEW MOVITRAC
//COPYRIGHT:    (C) 2004  BUHLER AG, CH-9240 UZWIL, SWITZERLAND
//
//PRODUCT:      SSA
//
//TITLE:        SEW MOVITRAC Frequency Inverter Profibus Communication
//
//--------------------------------------------------------------------------------
//
//IDENT:         AUTHOR:             DEPT:                            DATE:
//
//FB1812.2.0     M.Wedler            AEB41                            13-Okt-2008
//               2nd Release
//FB1811.1.0     A.Egli              CT3                              13-Jul-2007
//               1st Release
//
//--------------------------------------------------------------------------------
//
//PURPOSE: 
//
//MANUAL : 
//
//RESTRICTIONS: 
//
//--------------------------------------------------------------------------------
//
AUTHOR : MW
FAMILY : STD
VERSION : 0.0
VAR
  InValuePC : INT ;	//Setpoint value 1 in [0.01 %]
  InEnableRev : BOOL ;
  InEnableFwd : BOOL ;
  CmdFaultReset : BOOL ;
  OutRunningRev : BOOL ;	//Feedback for element motor
  OutRunningFwd : BOOL ;	//Feedback for element motor
  OutFault : BOOL ;	//Feedback for element motor
  MotorStStopped : BOOL ;	//Motor has come to a standstill after stopping time
  Spare : BOOL ;
  OutValuePC : INT ;	//Aktuel value 1 in [0.01 %]
  Input : STRUCT
   StateWord_1 : STRUCT 	//Statuswort MOVIDRIVE
    STATE_WORD_BIT_8 : BOOL ;	//Geraetezustand / Fehelr-Nummer
    STATE_WORD_BIT_9 : BOOL ;	//Geraetezustand / Fehelr-Nummer
    STATE_WORD_BIT_10 : BOOL ;	//Geraetezustand / Fehelr-Nummer
    STATE_WORD_BIT_11 : BOOL ;	//Geraetezustand / Fehelr-Nummer
    STATE_WORD_BIT_12 : BOOL ;	//Geraetezustand / Fehelr-Nummer
    STATE_WORD_BIT_13 : BOOL ;	//Geraetezustand / Fehelr-Nummer
    STATE_WORD_BIT_14 : BOOL ;	//Geraetezustand / Fehelr-Nummer
    STATE_WORD_BIT_15 : BOOL ;	//Geraetezustand / Fehelr-Nummer
    ENDSTUFE_FREIGEGEBEN : BOOL ;	//0=Endstufe gesperrt                 1=Endstufe freigegeben
    BETRIEBSBEREIT : BOOL ;	//0=Umrichter nicht betriebsbereit    1=Umrichter betriebsbereit
    PA_DATEN_FREIGEGEBEN : BOOL ;	//0=PA-Daten gesperrt                 1=PA-Daten freigegeben
    AKTUELL_INTEGRATORSATZ : BOOL ;	//0=Integrator 1                      1=Integrator 2
    AKTUELL_PARAMETERSATZ : BOOL ;	//0=Parametersatz 1                   1=Parametersatz 2
    STOERUNG_WARNUNG : BOOL ;	//0=keine Störung/Warnung             1=Störung/Warnung
    LS_RECHTS_AKTIV : BOOL ;	//1=Endschalter RECHTS betaetigt -> Drehrichtung RECHTS gesperrt
    LS_LINKS_AKTIV : BOOL ;	//1=Endschalter LINKS betaetigt -> Drehrichtung LINKS gesperrt
   END_STRUCT ;
   ActualValue01 : INT ;	//Hauptistwert / Prozessdaten PD2
   ActualValue02 : INT ;	//Prozessdaten PD3
   ActualValue03 : INT ;	//Prozessdaten PD4
   ActualValue04 : INT ;	//Prozessdaten PD5
   ActualValue05 : INT ;	//Prozessdaten PD6
  END_STRUCT ;
  Output : STRUCT
   ControlWord_1 : STRUCT 	//Steuerwort MOVIDRIVE
    CONTROL_WORD_BIT_8 : BOOL ;	//Reserviert für Zusatzfuktionen = "0"
    CONTROL_WORD_BIT_9 : BOOL ;	//Reserviert für Zusatzfuktionen = "0"
    CONTROL_WORD_BIT_10 : BOOL ;	//Reserviert für Zusatzfuktionen = "0"
    CONTROL_WORD_BIT_11 : BOOL ;	//Reserviert für Zusatzfuktionen = "0"
    CONTROL_WORD_BIT_12 : BOOL ;	//Reserviert für Zusatzfuktionen = "0"
    CONTROL_WORD_BIT_13 : BOOL ;	//Reserviert für Zusatzfuktionen = "0"
    CONTROL_WORD_BIT_14 : BOOL ;	//Reserviert für Zusatzfuktionen = "0"
    CONTROL_WORD_BIT_15 : BOOL ;	//Reserviert für Zusatzfuktionen = "0"
    REGLERSPERRE : BOOL ;	//0=Freigabe                          1=Regler sperren, Bremse aktivieren
    FREIGABE_SCHNELLSTOPP : BOOL ;	//0=Schnellstopp                      1=Freigabe
    FREIGABE_HALT : BOOL ;	//0=Halt an Integrator/Prozess-Rampe  1=Freigabe
    HALTEREGELUNG : BOOL ;	//0=Halteregelung nicht aktiv         1=Halteregelung aktiv
    INTEGRATOR : BOOL ;	//0=Integrator 1                      1=Integrator 2
    PARAMETERSATZ : BOOL ;	//0=Parametersatz 1                   1=Parametersatz 2
    RESET : BOOL ;	//0=nicht aktiv                       1=Fehler quittieren
    RESERVE_BIT_7 : BOOL ;	//Reserviert für Zusatzfuktionen = "0"
   END_STRUCT ;
   SetpointValue01 : INT ;	//Hauptsollwert / Prozessdaten PD2
   SetpointValue02 : INT ;	//Prozessdaten PD3
   SetpointValue03 : INT ;	//Prozessdaten PD4
   SetpointValue04 : INT ;	//Prozessdaten PD5
   SetpointValue05 : INT ;	//Prozessdaten PD6
  END_STRUCT ;
  Par : STRUCT
   spare1 : INT ;
   spare2 : INT ;
   spare3 : INT ;
   ParMOVITRAC : BOOL ;
   ParSinamics : BOOL ;
   ParMicromaster : BOOL ;
   ParABB : BOOL ;
   ParNord : BOOL ;
   ParDanfoss : BOOL ;
   ParIOByteNo : INT ;
  END_STRUCT ;
END_VAR
VAR_TEMP
  tmpAddrDB : INT ;
  tmpAddrIO : DINT ;
  tmpAddrInputFU : DINT ;
  tmpAddrOutputFU : DINT ;
END_VAR
BEGIN
NETWORK
TITLE = Calculate Address of Inverter
      L     #Par.ParIOByteNo;
      SLD   3;
      T     #tmpAddrIO;
      L     P##Input;
      L     DW#16#FFFFFF;
      AD;
      TAR2;
      +D;
      T     #tmpAddrInputFU;
      L     P##Output;
      L     DW#16#FFFFFF;
      AD;
      TAR2;
      +D;
      T     #tmpAddrOutputFU;
NETWORK
TITLE = Prepare Commands for Inverter SEW MOVITRAC
      AN    #Par.ParMOVITRAC;
      JC    MDJ0;
//- Prepare steuerword
      A     #Input.StateWord_1.STATE_WORD_BIT_15;
      =     #Output.ControlWord_1.FREIGABE_SCHNELLSTOPP;
      A     #InEnableFwd;
      O     #InEnableRev;
      =     #Output.ControlWord_1.REGLERSPERRE;
NETWORK
TITLE = Prepare setpoint value
//Motor nominal speed:
//C000H = -16384Dez = -100.0% (direction left)
//4000H = +16384Dez = +100.0% (direction right)
      L     #OutValuePC;
      ITD;
      DTR;
      L     1.638400e+00;
      *R;
      RND;
      A     #InEnableRev;
      JCN   tsp;
      NEGD;
tsp:  T     #Output.SetpointValue01;
NETWORK
TITLE = Communication to Inverter SEW MOVITRAC               
      CALL  "Standard_MC07" (
           DRIVE_IO_ADDRESS         := #Par.ParIOByteNo,
           ENABLE_RAPID_STOP        := #Output.ControlWord_1.FREIGABE_SCHNELLSTOPP,
           ENABLE                   := #Output.ControlWord_1.REGLERSPERRE,
           RESET                    := #CmdFaultReset,
           SETPOINT_SPEED           := #Output.SetpointValue01,
           RAMP                     := 10000,
           COMMUNICATION_OK         := #Input.StateWord_1.STATE_WORD_BIT_15,
           INVERTER_READY           := #Input.StateWord_1.BETRIEBSBEREIT,
           FAULT_OF_AXIS            := #Input.StateWord_1.STOERUNG_WARNUNG,
           FAULT_NO                 := #Input.ActualValue05,
           ACTUAL_SPEED             := #Input.ActualValue01,
           OUTPUT_CURRENT           := #Input.ActualValue02);
NETWORK
TITLE = Set State of Inverter SEW MOVITRAC
//- Feedback for motor
      A     #Input.StateWord_1.BETRIEBSBEREIT;
      AN    #Input.StateWord_1.STOERUNG_WARNUNG;
      A     #InEnableRev;
      =     #OutRunningRev;
      A     #Input.StateWord_1.BETRIEBSBEREIT;
      AN    #Input.StateWord_1.STOERUNG_WARNUNG;
      A     #InEnableFwd;
      =     #OutRunningFwd;
      A     #Input.StateWord_1.STOERUNG_WARNUNG;
      =     #OutFault;
NETWORK
TITLE = Prepare actual value
//Motor nominal speed:
//C000H = -16384Dez = -100.0% (direction left)
//4000H = +16384Dez = +100.0% (direction right)
      L     #Input.ActualValue01;
      ITD;
      DTR;
      ABS;
      L     1.638400e+00;
      /R;
      RND;
      T     #InValuePC;
NETWORK
TITLE =
      A     #CmdFaultReset;
      R     #CmdFaultReset;
NETWORK
TITLE =
MDJ0: NOP   0;
      BE;
END_FUNCTION_BLOCK

// FC 34: know-how protected block, not included

// FC 35: know-how protected block, not included

FUNCTION "Standard_MC07" : VOID	// FC 130
//Dieses Programmbeispiel zeigt nur die prinzipielle Vorgehensweise.
//Für fehlerhafte Programmfunktionen und deren Folgen
//kann weder eine juristische, noch irgendeine Haftung übernommen werden!
AUTHOR : GE-AT
FAMILY : PROFIBUS
NAME : MC07_UFP
VERSION : 1.0
VAR_INPUT
  DRIVE_IO_ADDRESS : INT ;
  ENABLE_RAPID_STOP : BOOL ;
  ENABLE : BOOL ;
  RESET : BOOL ;
  SETPOINT_SPEED : INT ;
  RAMP : INT ;
END_VAR
VAR_OUTPUT
  COMMUNICATION_OK : BOOL ;	//SFC14/SFC15: Return Value = 0
  INVERTER_READY : BOOL ;
  FAULT_OF_AXIS : BOOL ;
  FAULT_NO : INT ;
  ACTUAL_SPEED : INT ;
  OUTPUT_CURRENT : INT ;
END_VAR
VAR_TEMP
  PI : STRUCT
   STATUS : BYTE ;
   ENABLE_OUTPUT_STAGE : BOOL ;
   INVERTER_READY : BOOL ;
   PO_DATA_ENABLE : BOOL ;
   STW_Bit_3 : BOOL ;
   STW_Bit_4 : BOOL ;
   ERROR : BOOL ;
   STW_Bit_6 : BOOL ;
   STW_Bit_7 : BOOL ;
   ACTUAL_SPEED : INT ;
   OUTPUT_CURRENT : INT ;
  END_STRUCT ;
  PO : STRUCT
   DIRECTION_MOTOR_POTI : BOOL ;
   MOTOR_POTI_UP : BOOL ;
   MOTOR_POTI_DOWN : BOOL ;
   FIXED_INTERNAL_SETPOINTS : BOOL ;
   FIXED_INTERNAL_SETP_1 : BOOL ;
   FIXED_SETP_SWITCHOVER : BOOL ;
   CTW_Bit_14 : BOOL ;
   CTW_Bit_15 : BOOL ;
   CONTR_INHIBIT : BOOL ;
   RAPID_STOP : BOOL ;
   STOP : BOOL ;
   CTW_Bit_3 : BOOL ;
   CTW_Bit_4 : BOOL ;
   CTW_Bit_5 : BOOL ;
   RESET_FAULT : BOOL ;
   CTW_Bit_7 : BOOL ;
   SETPOINT_SPEED : INT ;
   RAMP : INT ;
  END_STRUCT ;
  RETURNCODE_SFC14 : INT ;
  RETURNCODE_SFC15 : INT ;
  ADDR : WORD ;
END_VAR
BEGIN
NETWORK
TITLE = Prozeßeingangsdaten aufbereiten
      L     #DRIVE_IO_ADDRESS;	//Adresse von "INT" nach "WORD" wandeln
      T     #ADDR;
      CALL  "DPRD_DAT" (
           LADDR                    := #ADDR,
           RET_VAL                  := #RETURNCODE_SFC14,
           RECORD                   := #PI);	//konsistente Daten eines DP-Normslaves lesen / Peripherieadresse => Hardwarekonfig. / <> 0 => ein Fehler ist während der Bearbeitung aufgetreten / Zielbereich für die gelesenen Nutzdaten.
      L     #RETURNCODE_SFC14;
      L     0;
      <>I;	//Tritt während der Abarbeitung der SFC ein Fehler auf,
      JC    END;	//so wird die Funktion verlassen => NW7
      L     #PI.ACTUAL_SPEED;
      T     #ACTUAL_SPEED;
      L     #PI.OUTPUT_CURRENT;
      L     10;	//Anpassung 1 digit = 0.1% In auf 1% In
      /I;
      T     #OUTPUT_CURRENT;
      A     #PI.INVERTER_READY;
// MW 2008.10.25
      A     #PI.PO_DATA_ENABLE;
      =     #INVERTER_READY;
      A     #PI.ERROR;
      =     #FAULT_OF_AXIS;
NETWORK
TITLE = Fehlermeldungen auswerten/rangieren
//Ist das Fehlerbit gesetzt, so wird die Fehlernummer ausgegeben.
//Liegt kein Fehler vor, so wird eine Null ausgegeben.
      A(;
      A     #PI.ERROR;
      JNB   _001;
      L     #PI.STATUS;
      T     #FAULT_NO;
      SET;
      SAVE;
      CLR;
_001: A     BR;
      );
      NOT;
      JNB   _002;
      L     0;
      T     #FAULT_NO;
_002: NOP   0;
NETWORK
TITLE = Prozeßausgangsdaten: Freigabe / Schnellstopp rangieren
      A     #ENABLE_RAPID_STOP;
      =     #PO.RAPID_STOP;
NETWORK
TITLE = Prozeßausgangsdaten: Regler-Freigabe
      A     #ENABLE;
      =     #PO.STOP;
NETWORK
TITLE = Fault_Reset
      A     #RESET;
      =     #PO.RESET_FAULT;
NETWORK
TITLE = Prozeßausgangsdaten aufbereiten
      SET;	//Rücksetzen aller nicht verwendeten Steuerwort-Bits
      R     #PO.CONTR_INHIBIT;
      R     #PO.CTW_Bit_3;
      R     #PO.CTW_Bit_4;
      R     #PO.CTW_Bit_5;
      R     #PO.CTW_Bit_7;
      R     #PO.DIRECTION_MOTOR_POTI;
      R     #PO.MOTOR_POTI_UP;
      R     #PO.MOTOR_POTI_DOWN;
      R     #PO.FIXED_INTERNAL_SETPOINTS;
      R     #PO.FIXED_INTERNAL_SETP_1;
      R     #PO.FIXED_SETP_SWITCHOVER;
      R     #PO.CTW_Bit_14;
      R     #PO.CTW_Bit_15;
      L     #SETPOINT_SPEED;
      T     #PO.SETPOINT_SPEED;
      L     #RAMP;
      T     #PO.RAMP;
      CALL  "DPWR_DAT" (
           LADDR                    := #ADDR,
           RECORD                   := #PO,
           RET_VAL                  := #RETURNCODE_SFC15);	//Daten konsistent auf einen DP-Normslave schreiben / Peripherieadresse => Hardwarekonfig. / Quellbereich für die zu schreibenden Nutzdaten / <> 0 => ein Fehler ist während der Bearbeitung aufgetreten
      L     #RETURNCODE_SFC15;	//Tritt während der Abarbeitung des SFCs ein Fehler auf, 
      L     0;
      <>I;
      JC    END;	//so wird die Funktion verlassen. => NW7
      =     #COMMUNICATION_OK;
      BEU;	//Ende der Funktion
NETWORK
TITLE = Kommunikationsfehler auswerten
//Ist die Abarbeitung der SFCs fehlerhaft, so werden alle Ausgänge der Funktion 
//abgelöscht
//
END:  L     0;
      T     #FAULT_NO;
      T     #ACTUAL_SPEED;
      T     #OUTPUT_CURRENT;
      SET;
      R     #COMMUNICATION_OK;
      R     #FAULT_OF_AXIS;
      R     #INVERTER_READY;
END_FUNCTION

FUNCTION "Test_Simuli" : VOID	// FC 999
AUTHOR : MW
VERSION : 0.1
BEGIN
NETWORK
TITLE =
      AN    DB50.DBX 33.0;
      BEC;
NETWORK
TITLE = ABB
// Statuswort
      L     W#16#207;
      T     IW 1000;	// StateWord_1
      T     IW 1040;	// StateWord_1
      T     IW 1080;	// StateWord_1
      T     IW 1120;	// StateWord_1
      T     IW 1160;	// StateWord_1
      T     IW 1200;	// StateWord_1
      T     IW 1220;	// StateWord_1
// Istwert = Sollwert
      L     QW 1002;	// SetpointValue01
      T     IW 1002;	// ActualValue01
      L     QW 1042;	// SetpointValue01
      T     IW 1042;	// ActualValue01
      L     QW 1082;	// SetpointValue01
      T     IW 1082;	// ActualValue01
      L     QW 1122;	// SetpointValue01
      T     IW 1122;	// ActualValue01
      L     QW 1162;	// SetpointValue01
      T     IW 1162;	// ActualValue01
      L     QW 1202;	// SetpointValue01
      T     IW 1202;	// ActualValue01
      L     QW 1222;	// SetpointValue01
      T     IW 1222;	// ActualValue01
NETWORK
TITLE = NORDAC
//      L     W#16#147F                   // Start direction left 
//      L     W#16#1007                   // Feedback started direction left
//      L     W#16#C7F                    // Start direction right
//      L     W#16#807                    // Feedback started direction right
// Statuswort
      L     QW 1020;	// ControlWord_1
      L     W#16#147F;	// Start direction left 
      ==I;
      L     W#16#1007;	// Feedback started direction left
      JC    N001;
      L     QW 1020;	// ControlWord_1
      L     W#16#C7F;	// Start direction right
      ==I;
      L     W#16#807;	// Feedback started direction right
      JC    N001;
      L     W#16#3;	// Feedback stopped                 
N001: T     IW 1020;	// StateWord_1
      L     QW 1060;	// ControlWord_1
      L     W#16#147F;	// Start direction left 
      ==I;
      L     W#16#1007;	// Feedback started direction left
      JC    N002;
      L     QW 1060;	// ControlWord_1
      L     W#16#C7F;	// Start direction right
      ==I;
      L     W#16#807;	// Feedback started direction right
      JC    N002;
      L     W#16#3;	// Feedback stopped                 
N002: T     IW 1060;	// StateWord_1
      L     QW 1100;	// ControlWord_1
      L     W#16#147F;	// Start direction left 
      ==I;
      L     W#16#1007;	// Feedback started direction left
      JC    N003;
      L     QW 1100;	// ControlWord_1
      L     W#16#C7F;	// Start direction right
      ==I;
      L     W#16#807;	// Feedback started direction right
      JC    N003;
      L     W#16#3;	// Feedback stopped                 
N003: T     IW 1100;	// StateWord_1
      L     QW 1140;	// ControlWord_1
      L     W#16#147F;	// Start direction left 
      ==I;
      L     W#16#1007;	// Feedback started direction left
      JC    N004;
      L     QW 1140;	// ControlWord_1
      L     W#16#C7F;	// Start direction right
      ==I;
      L     W#16#807;	// Feedback started direction right
      JC    N004;
      L     W#16#3;	// Feedback stopped                 
N004: T     IW 1140;	// StateWord_1
      L     QW 1180;	// ControlWord_1
      L     W#16#147F;	// Start direction left 
      ==I;
      L     W#16#1007;	// Feedback started direction left
      JC    N005;
      L     QW 1180;	// ControlWord_1
      L     W#16#C7F;	// Start direction right
      ==I;
      L     W#16#807;	// Feedback started direction right
      JC    N005;
      L     W#16#3;	// Feedback stopped                 
N005: T     IW 1180;	// StateWord_1
      L     QW 1240;	// ControlWord_1
      L     W#16#147F;	// Start direction left 
      ==I;
      L     W#16#1007;	// Feedback started direction left
      JC    N006;
      L     QW 1240;	// ControlWord_1
      L     W#16#C7F;	// Start direction right
      ==I;
      L     W#16#807;	// Feedback started direction right
      JC    N006;
      L     W#16#3;	// Feedback stopped                 
N006: T     IW 1240;	// StateWord_1
// Istwert = Sollwert
      L     QW 1022;	// SetpointValue01
      T     IW 1022;	// ActualValue01
      L     QW 1062;	// SetpointValue01
      T     IW 1062;	// ActualValue01
      L     QW 1102;	// SetpointValue01
      T     IW 1102;	// ActualValue01
      L     QW 1142;	// SetpointValue01
      T     IW 1142;	// ActualValue01
      L     QW 1182;	// SetpointValue01
      T     IW 1182;	// ActualValue01
      L     QW 1242;	// SetpointValue01
      T     IW 1242;	// ActualValue01
NETWORK
TITLE = Danfoss
//MW 2008.09.02
// Statuswort
      L     W#16#F07;
      T     IW 1300;	// StateWord_1
      T     IW 1310;	// StateWord_1
// Istwert = Sollwert
      L     QW 1302;	// SetpointValue01
      A     DB198.DBX 828.3;
      O     DB198.DBX 828.4;
      JC    ew;
      L     0;
ew:   T     IW 1302;	// ActualValue01
      L     QW 1312;	// SetpointValue01
      A     DB199.DBX 828.3;
      O     DB199.DBX 828.4;
      JC    Ew;
      L     0;
Ew:   T     IW 1312;	// ActualValue01
NETWORK
TITLE = Interface
NETWORK
TITLE =
      BE;
END_FUNCTION

FUNCTION FC 1010 : VOID
TITLE = Prozesszeit aus der CPU-Uhrzeit bilden
//  
//COPYRIGHT:    (C) 2003  Bühler GmbH D-38114 Braunschweig Deutschland
//
//PRODUCT:      GCS7
//
//TITLE:        Prozesszeit
//
//-------------------------------------------------------------------------
//
//IDENT:        AUTHOR:             DEPT:                       DATE:
//FC10.1B      J. Voss             AEB3                        12.10.05
//              T110 Verz Löschen Prozessminute 
//
//FC10.1A      J. Voss             AEB3                        23.09.03
//              1st Release 
//
//-------------------------------------------------------------------------
//
//PURPOSE:      Erfassen der Prozesszeit für eine Sektion aus der CPU Zeit        
//              Für bis zu 16 Sektionen
//              Benötigt DB mit entsprechender Struktur (DB10)
//
//RESTRICTIONS:    Benötigt einen DB mit zwei Feldern dt1 und dt2 im Format 
//                 DATE_AND_TIME und einem Feld Diff im Format TIME, sowie 
//                 für die Tage/Stunden/Minuten je ein Feld im Format INT
//                 Aufgerufen werden SFC_1 "READ_CLK" und FC34 SB_DT_DT
//-------------------------------------------------------------------------
//
//
AUTHOR : JV
VERSION : 0.1
BEGIN
NETWORK
TITLE =
//Bleibt frei
NETWORK
TITLE = in Arbeitsbereich kopieren
      L     "DB Prozesszeit".Zaehler;
      L     "DB Prozesszeit".Anzahl_Sektionen;
      >I;
      JCN   Copy;
      L     "DB Prozesszeit".ErsteSektion;
      T     "DB Prozesszeit".Zaehler;
      L     "DB Prozesszeit".ErsteSektion;
      L     1;
      -I;
      L     60;	// Länge pro Sektion
      *I;
      L     70;	// Start erste Sektion
      +I;
      T     "DB Prozesszeit".ZeigerLesenSchreiben;
Copy: NOP   0;
      CALL  FC 49 (
           $1                       := 1010,
           $2                       := "DB Prozesszeit".ZeigerLesenSchreiben,
           $3                       := 1010,
           $4                       := 10,
           $5                       := 60,
           $6                       := P#M 200.0);
NETWORK
TITLE = Prozesszeit ausrechnen
      CALL  SFC 1 (
           $1                       := "DB Prozesszeit".Arbeitsbereich.temp1,
           $2                       := "DB Prozesszeit".Arbeitsbereich.dt2);
      A     "DB Prozesszeit".Arbeitsbereich.Prozess_aktiv;	// Prozesszeit aktiv
      JC    end;
      CALL  SFC 1 (
           $1                       := "DB Prozesszeit".Arbeitsbereich.temp1,
           $2                       := "DB Prozesszeit".Arbeitsbereich);
end:  NOP   0;
      CALL  "SB_DT_DT" (
           $1                       := "DB Prozesszeit".Arbeitsbereich.dt2,
           $2                       := "DB Prozesszeit".Arbeitsbereich,
           $3                       := "DB Prozesszeit".Arbeitsbereich.Diff);
NETWORK
TITLE = Prozesszeit Minutenzaehler
// 
      A     "DB Prozesszeit".Arbeitsbereich.Prozess_aktiv;	// Prozesszeit aktiv
      L     S5T#1S;
      SF    T 110;	//  Verzögerung löschen Minuten
// 
      L     0;
      A     T 110;	//  Verzögerung löschen Minuten
      JCN   Nost;
      L     "DB Prozesszeit".Arbeitsbereich.Diff;
      L     L#60000;	// ms/min
      /D;
      T     MD 206;
      L     MW 208;
Nost: NOP   0;
      T     "DB Prozesszeit".Arbeitsbereich.Gesamtzeit_in_Minuten;	// Prozesszeit gesamt in Minuten
      NOP   0;
NETWORK
TITLE = Prozesszeit Tage, Stunden, Minuten ermitteln
// (network holds code this reader does not know; not shown)
NETWORK
TITLE = Zeitanzeigen für WinCC
// Tagesanzeige für Visu
      L     0;
      A     "DB Prozesszeit".Arbeitsbereich.Prozess_aktiv;	// Prozesszeit aktiv
      JCN   tDay;
      L     "DB Prozesszeit".Arbeitsbereich.Tage;
      L     1;
      +I;
tDay: NOP   0;
      T     "DB Prozesszeit".Arbeitsbereich.Visu_Tage;	// Anzeige Prozesstag (1 = 1. Tag)
// Stundenanzeige 0-24 für Visu
      L     0;
      A     "DB Prozesszeit".Arbeitsbereich.Prozess_aktiv;	// Prozesszeit aktiv
      JCN   tHur;
      L     "DB Prozesszeit".Arbeitsbereich.Stunden;
      T     MD 206;
      L     MW 208;
tHur: NOP   0;
      T     "DB Prozesszeit".Arbeitsbereich.Visu_StundenProTag;	// Anzeige Stunden pro Tag
// Minutenanzeige (0-59) nur fuer Visu
      L     0;
      A     "DB Prozesszeit".Arbeitsbereich.Prozess_aktiv;	// Prozesszeit aktiv
      JCN   tMin;
      L     "DB Prozesszeit".Arbeitsbereich.Minuten;
      T     MD 206;
      L     MW 208;
tMin: NOP   0;
      T     "DB Prozesszeit".Arbeitsbereich.Visu_MinutenProStunde;	// Anzeige Minuten pro Sunde
NETWORK
TITLE = Zeitpointer
//Hier werden Zeitpointer erzeugt, um andere Raster als Stundenrythmus zu erhalten
//
//  10 Minuten Raster
      L     "DB Prozesszeit".Arbeitsbereich.Diff;
      L     L#600000;	// Millisec/10 min
      /D;
      T     MD 200;
      L     MW 202;
      T     "DB Prozesszeit".Arbeitsbereich.Pointer_10min;
// 30 Minuten Raster
      L     "DB Prozesszeit".Arbeitsbereich.Diff;
      L     L#1800000;	// Millisec/30 min
      /D;
      T     MD 200;
      L     MW 202;
      T     "DB Prozesszeit".Arbeitsbereich.Pointer_30min;
//  90 Minuten Raster
      L     "DB Prozesszeit".Arbeitsbereich.Diff;
      L     L#2400000;	// Millisec/90 min
      /D;
      T     MD 200;
      L     MW 202;
      T     "DB Prozesszeit".Arbeitsbereich.Pointer_90min;
NETWORK
TITLE = zurück in die Sektion
// 
      CALL  FC 49 (
           $1                       := 1010,
           $2                       := 10,
           $3                       := 1010,
           $4                       := "DB Prozesszeit".ZeigerLesenSchreiben,
           $5                       := 60,
           $6                       := P#M 200.0);
      L     "DB Prozesszeit".Zaehler;
      L     1;
      +I;
      T     "DB Prozesszeit".Zaehler;	// Nächster Block
      L     "DB Prozesszeit".ZeigerLesenSchreiben;
      L     60;	// Länge pro Sektion
      +I;
      T     "DB Prozesszeit".ZeigerLesenSchreiben;	// 
NETWORK
TITLE =
      BE;
END_FUNCTION

FUNCTION "Act_Value_LogConvert" : VOID	// FC 1045
TITLE = Log: Message Converter for LOG Entry
//COPYRIGHT:     (C) 1996 BY  BUEHLER LTD. 
//                            CH-9240 UZWIL  SWITZERLAND
//
//PRODUCT:      GCS7 
//
//TITLE:        Message Converter for LOG Entry
//
//--------------------------------------------------------------------------
//
//IDENT:        AUTOR:              DEPT:                       DATE:
//
//FC45.1.2      A. Egli             CT3                         04.03.2003
//              Redesign, M11.2
//FC45.1B       A. Egli             CT3                         26.03.1999
//              Special format for MELE: MsgType>=7000
//FC45.1A       S. Kalberer         AEE61                       27-Sep-1996
//              1st Release in S7, converted from FX251.2A
//
//--------------------------------------------------------------------------
//
//PURPOSE:       DATA-CONVERT FOR PRINTER PER LOG WITH PC
//
//RESTRICTIONS:  S7
//
//--------------------------------------------------------------------------
//
AUTHOR : EA
FAMILY : GCS7LL
NAME : MECONV
VERSION : 0.0
VAR_INPUT
  ObjectNo : INT ;	//Is used for communication with PC
  MsgType : INT ;	//Is used for message translation
  ClassMsgTxt : WORD ;	//Contains MessageClass and MessageTextNumber
  OType : INT ;	//Object Type
END_VAR
VAR_TEMP
  tmpHeader : WORD ;
  tmpPara2 : WORD ;
  tmpObjectNo : WORD ;
  tmpLineNo : WORD ;
  tmpMsgType : WORD ;
  tmpGr : INT ;
  tmpIndex : INT ;
END_VAR
BEGIN
NETWORK
TITLE =  MESSAGE
//Standard GCS90
      L     #ObjectNo;	// Change type INT --> WORD
      T     #tmpObjectNo;
      L     #ClassMsgTxt;	// Load: HighByte= Class ¦ Low Byte= TextNo (8 Bit)
      SRW   8;	// Delete TextNo
      SLW   5;
      +     13;	// add MessageFormatNo
      T     #tmpHeader;	//-> Header=Format := Class ¦ MsgFormatNo
      L     #ClassMsgTxt;	// Load: HighByte= Class ¦ Low Byte= TextNo (8 Bit)
      L     2#11111111;	// Delete Class
      AW;
      L     #MsgType;
      SLW   8;
      OW;
      T     #tmpPara2;	//-->Para2 := MsgType ¦ TextNo
      L     MB 14;
      T     #tmpLineNo;
      L     #MsgType;
      T     #tmpMsgType;
      A     M 11.2;
      JC    EQ00;
      CALL  FC 46 (
           $1                       := 5,
           $2                       := #tmpHeader,
           $3                       := #tmpObjectNo,
           $4                       := #tmpPara2,
           $5                       := #tmpLineNo,
           $6                       := #tmpMsgType,
           $7                       := 0,
           $8                       := 0,
           $9                       := 0,
           $10                      := 0,
           $11                      := 0,
           $12                      := 0,
           $13                      := 0);	//---Call Message Entry--- /  Queue DB Number                 /  Format /  ObjectNumber /  MsgType ¦ TextNo /  Line /  MsgType S7 /  not used  /  not used  /  not used  /  not used  /  not used  /  not used  /  not used
EQ00: NOP   0;
NETWORK
TITLE = End of Block
END_FUNCTION

FUNCTION "SSA_MH_LogEntry_ActValue" : VOID	// FC 1046
TITLE = Log: Message Entry
//COPYRIGHT:    (C) 1996 BY  BUEHLER LTD. 
//                           CH-9240 UZWIL  SWITZERLAND
//
//PRODUCT:      GCS7
//
//TITLE:        Entry in QUEUE for Actual Values to PC for Trace 
//
//-------------------------------------------------------------------------
//
//IDENT:        AUTHOR:             DEPT:                       DATE:
//
//
//FC1046.1A     S. Jennermann       AEB2                        7-Dec-2004
//              1st Release in S7, converted from FB46.2A
//
//-------------------------------------------------------------------------
//
//PURPOSE:      used in MT Plants               
//
//RESTRICTIONS: S7
//                                                          
//
//
//-------------------------------------------------------------------------
//
//        MESSAGE ENTRY               
//   +------------------------+   
// ->¦ DBNumber               ¦           LOG-DB
//   +------------------------+
//
AUTHOR : EA
FAMILY : GCS7SYS
NAME : MESENTRY
VERSION : 2.0
VAR_INPUT
  DBNumber : INT ;	//Queue DB-Number
END_VAR
VAR_TEMP
  tmpQueueDB : INT ;
  tmpHeader : WORD ;
  tmpCnt : WORD ;	//temp loop counter
  tmpSourceAddress : DWORD ;	//temp Source Address
  tmpBlockLength : DWORD ;	//temp Message BlockLength
  tmpEndOfQueue : WORD ;
  tmpOpenDB : INT ;
  tmpBytePrev : INT ;
  tmpMsgActive : BOOL ;
END_VAR
BEGIN
NETWORK
TITLE =  SAVE INPUT 
//---Save Input Parameter into temp variables
      L     #DBNumber;
      T     #tmpQueueDB;
      OPN   DB [#tmpQueueDB];
      L     DBW 4;	// ParByteLenghtUDT
      T     #tmpBlockLength;
//-- Init ---
      L     DBW 8;	// VarNrOfMsgInQueue
      L     0;
      <>I;
      JC    T0;	// Init Read Write Pointer
      L     DBW 16;	// -> ParStartFIFO
      T     DBW 10;	// -> varDWwrite
      T     DBW 12;	// -> varDWread
// 
T0:   L     DBW 10;	// varDWwrite
      L     DBW 16;	// -> ParStartFIFO
      >D;
      JC    T2;
      T     DBW 10;	// -> varDWwrite
T2:   L     DBW 12;	// varDWread
      L     DBW 16;	// -> ParStartFIFO
      >D;
      JC    T3;
      T     DBW 12;	// -> varDWread
T3:   L     DBW 6;	// ParMaxNrOfMsg
      L     #tmpBlockLength;
      *I;
      L     DBW 16;	// -> ParStartFIFO
      +I;	// --> Address end of queue
      T     #tmpEndOfQueue;
      L     DBW 6;	// ParMaxNrOfMsg 
NETWORK
TITLE =  Queue is full 
      L     DBW 6;	// ParMaxNrOfMsg 
      L     DBW 8;	// VarNrOfMsgInQueue
      <=I;
      JC    out;
NETWORK
TITLE = Test Queue full
//IF THERE IS ENOUGH PLACE FOR TWO MESSAGES AT LEAST
//  THEN
//    PUT PRINTORDER INTO WQ
      L     DBW 6;	//ParMaxNrOfMsg
      +     -1;
      L     DBW 8;	//VarNrOfMsgInQueue
      <=I;
      JC    FULL;
NETWORK
TITLE = Store Message in queue
//----Write Message in LOG-queue
      CALL  FC 49 (
           $1                       := #tmpQueueDB,
           $2                       := P#DBX 20.0,
           $3                       := #tmpQueueDB,
           $4                       := P#DBX 10.0,
           $5                       := P#DBX 4.0,
           $6                       := P#DBX 0.0);	// input Message /  Write pointer
      JU    NX06;
NETWORK
TITLE =  SET "WAITING QUEUE FULL"
//IF WAITING QUEUE FULL UNLESS ONE PLACE AND NO ERROR SET
//  THEN
//    SET INTERNAL MESSAGE
//    SET ERROR INPUT
FULL: NOP   0;
      CALL  FC 49 (
           $1                       := #tmpQueueDB,
           $2                       := P#DBX 18.0,
           $3                       := #tmpQueueDB,
           $4                       := P#DBX 10.0,
           $5                       := P#DBX 4.0,
           $6                       := P#DBX 0.0);	// Message full /  Write pointer
NETWORK
TITLE =  EPILOG
NX06: L     DBW 10;	// VarDWwrite
      L     #tmpBlockLength;
      +I;
      T     DBW 10;	// --> VarDWWrite
      A(;
      L     DBW 10;	// --> VarDWWrite
      L     #tmpEndOfQueue;
      <D;
      );
      JC    L002;
      L     DBW 16;	// PaStartFIFO
      T     DBW 10;	// --> VarDWWrite
L002: L     DBW 8;	// VarNrOfMsgInQueue
      +     1;
      T     DBW 8;	//-->VarNrOfMsgInQueue
out:  NOP   0;
      L     DBW 8;	// VarNrOfMsgInQueue
      L     0;
      ==I;
      JC    End;
      L     1;
End:  T     DBW 58;	// PC.NrOfMessageInQueue
END_FUNCTION

FUNCTION "SSA_MH_LogCtrl_ActValue" : VOID	// FC 1047
TITLE = Log: Read Queue Message
//COPYRIGHT:    (C) 1996 BY  BUEHLER LTD. 
//                           CH-9240 UZWIL  SWITZERLAND
//
//PRODUCT:      GCS7
//
//TITLE:        READ from QUEUE for GCS90-Upper-Level
//
//-------------------------------------------------------------------------
//
//IDENT:        AUTHOR:              DEPT:                       DATE:
//
//FC47.2.0      A.Egli               CT3                         14-Jul-2004
//              CmdAddFisrt
//FC47.1A       S. Kalberer          AEE61                       4-Dec-1996
//              1st Release in S7, converted from FB47.2A
//
//-------------------------------------------------------------------------
//
//PURPOSE:      MANUAL : see [CTRxxMAN]
//              This function reads 1 .. max. 4 print-orders out of the 
//              waiting-queue to set ready at the PC-Interface
//
//RESTRICTIONS: S7
//              Only for message administration on PC
//
//-------------------------------------------------------------------------
//
AUTHOR : EA
FAMILY : GCS7SYS
NAME : MESSFORM
VERSION : 2.0
VAR_INPUT
  DBNumber : INT ;	//Queue DB-Number
END_VAR
VAR_TEMP
  tmpDBNumber : INT ;	//Input Queue-DB
  tmpCnt : WORD ;	//temp loop counter
  tmpSourceAddress : DWORD ;	//temp Source Address
  tmpDestAddress : DWORD ;	//temp Target Address
  tmpTxtBufferPtr : DWORD ;	//ASA Textbuffer Pointer
  tmpBlockLength : WORD ;	//temp Message BlockLength
  tmpEndOfQueue : INT ;
END_VAR
BEGIN
NETWORK
TITLE =  MESSAGE-FORM
NETWORK
TITLE =  ADDRESS/LENGTH QUEUE
      L     #DBNumber;
      T     #tmpDBNumber;
      OPN   DB [#tmpDBNumber];	//>> CALL QUEUE-DB
      L     DBW 4;	// ParByteLengtMessage
      T     #tmpBlockLength;
NETWORK
TITLE =  CONFIGURATION TEST
      AN    DBX 46.7;	// CmdResetLog
      JC    L002;	// 
      R     DBX 46.7;	// CmdResetLog
      L     DBW 16;	// ParStartFIFO
      T     DBW 10;	// -> varDWwrite
      T     DBW 12;	// -> varDWread
      L     0;	// 
      T     DBW 8;	// VarNrOfMsgInQueue
      T     DBW 56;	// HskPLCtoPC
L002: L     DBW 10;	// varDWwrite
      L     DBW 16;	// ParStartFIFO
      >I;
      JC    T2;
      T     DBW 10;	// -> varDWwrite
T2:   L     DBW 12;	// varDWread
      L     DBW 16;	// ParStartFIFO
      >D;
      JC    T3;
      T     DBW 12;	// -> varDWread
T3:   L     DBW 6;	// ParMaxNrOfMsg
      L     #tmpBlockLength;
      *I;
      L     DBW 16;	// ParStartFIFO
      +I;	// --> Address end of queue
      T     #tmpEndOfQueue;
      L     DBLG;
      >D;
      JC    ERRO;	//-->(ERROR= DB to small)
      L     #tmpEndOfQueue;
      L     #tmpBlockLength;
      -I;
      L     DBW 12;	//  
      <D;	// varDWread
      JC    ERRO;	// -->ERROR= Read Pointer
      JU    NX04;
ERRO: BEU;	// ERROR QUEUE
NETWORK
TITLE =  TEST HANDSHAKE
NX04: L     DBW 44;	//---par_PC_connection[2..1]
      L     DBW 44;	//[2.0]
      SLD   4;	//[2.0]
      OW;	//[2.0]
      L     DBW 56;	// HskPLCtoPC
      AW;
      L     DBW 46;	// inf_control (PC Off-Line)
      INVI;	// Complement 1
      AW;
      T     DBW 56;	// HskPLCtoPC
      A     DBX 49.0;	// HskPC1toPLC.MsgDone
      R     DBX 49.0;	// HskPC1toPLC.MsgDone
      R     DBX 57.0;	// HskPLCtoPC.MsgForPC1
      A     DBX 49.1;	//[2.0] HskPC1toPLC.MsgDone
      R     DBX 49.1;	//[2.0] HskPC1toPLC.MsgDone
      R     DBX 57.4;	//[2.0] HskPLCtoPC.MsgForPC1
      A     DBX 51.0;	// HskPC2toPLC.MsgDone
      R     DBX 51.0;	// HskPC2toPLC.MsgDone
      R     DBX 57.1;	// HskPLCtoPC.MsgForPC2
      A     DBX 51.1;	//[2.0] HskPC2toPLC.MsgDone
      R     DBX 51.1;	//[2.0] HskPC2toPLC.MsgDone
      R     DBX 57.5;	//[2.0] HskPLCtoPC.MsgForPC2
      A     DBX 53.0;	// HskPC3toPLC.MsgDone
      R     DBX 53.0;	// HskPC3toPLC.MsgDone
      R     DBX 57.2;	// HskPLCtoPC.MsgForPC3
      A     DBX 53.1;	//[2.0] HskPC3toPLC.MsgDone
      R     DBX 53.1;	//[2.0] HskPC3toPLC.MsgDone
      R     DBX 57.6;	//[2.0] HskPLCtoPC.MsgForPC3
      A     DBX 55.0;	// HskPC4toPLC.MsgDone
      R     DBX 55.0;	// HskPC4toPLC.MsgDone
      R     DBX 57.3;	// HskPLCtoPC.MsgForPC4
      A     DBX 55.1;	//[2.0] HskPC4toPLC.MsgDone
      R     DBX 55.1;	//[2.0] HskPC4toPLC.MsgDone
      R     DBX 57.7;	//[2.0] HskPLCtoPC.MsgForPC4
      L     0;	//---Handshake is read
      L     DBW 56;	// HskPLCtoPC
      <>I;	// message not read
      BEC;
NETWORK
TITLE =  READ MESSAGE
      L     DBW 8;	// VarNoOfMsgInQueue
      L     0;
      ==I;
      BEC;
      CALL  FC 49 (
           $1                       := #tmpDBNumber,
           $2                       := P#DBX 12.0,
           $3                       := #tmpDBNumber,
           $4                       := P#DBX 2.0,
           $5                       := P#DBX 4.0,
           $6                       := P#DBX 0.0);	// Read Pointer /  ParByteReadQueuPC
      L     DBW 12;	// read Pointer
      L     #tmpBlockLength;
      +I;
      T     DBW 12;	// read Pointer
      L     #tmpEndOfQueue;
      <D;
      JC    L003;
      L     DBW 16;	// ParDWStartQueue
      T     DBW 12;	// read Pointer
L003: L     DBW 8;	// VarNrOfMsgInQueue
      +     -1;
      T     DBW 8;	//-->VarNrOfMsgInQueue
//---Send to PC -----
      L     DBW 44;	// ParPCconnection
      L     DBW 56;	// HskPLCtoPC
      OW;
      T     DBW 56;	// HskPLCtoPC
      S     DBX 41.0;	//---Set change-bit
END_FUNCTION

FUNCTION "SSA_MH_Increment_counter" : VOID	// FC 1048
TITLE = Incremental Counter
//COPYRIGHT:    (C) 1996 BY  BUEHLER LTD. 
//                           CH-9240 UZWIL  SWITZERLAND
//
//PRODUCT:      GCS7
//
//TITLE:        READ from QUEUE for GCS90-Upper-Level
//
//-------------------------------------------------------------------------
//
//IDENT:        AUTHOR:              DEPT:                       DATE:
//
//FC1048.1A     U. Kemmesies         AEB41                       7-Dec-2007
//              1st Release in S7
//
//-------------------------------------------------------------------------
//
//PURPOSE:      MANUAL : see [CTRxxMAN]
//              This function reads the two tracks from an incremental counter 
//              and give out the counter value
//
//RESTRICTIONS: S7
//              Only for message administration on PC
//
//-------------------------------------------------------------------------
//
VERSION : 0.1
VAR_INPUT
  Eingang1 : BOOL ;
  Eingang2 : BOOL ;
END_VAR
VAR_IN_OUT
  Zahler : UDT 20851;
END_VAR
BEGIN
NETWORK
TITLE = Inputs counter device
      AN    #Eingang1;	// Track A
      BLD   5;
      T     LD 2;
      TAK;	// Track B
      T     LD 6;
      L     P##Zahler;
      LAR1;	// Track A
      L     W [AR1,P#0.0];
      T     LW 0;
      OPN   DB [LW 0];
// 
      L     D [AR1,P#2.0];	// Track B
      LAR1;
      L     LD 6;
      L     LD 2;
      R      [AR1,P#6.0];
      BLD   5;
      T     LD 2;
      TAK;
      T     LD 6;
      L     P##Zahler;
      LAR1;
      L     W [AR1,P#0.0];
      T     LW 0;
      OPN   DB [LW 0];
      L     D [AR1,P#2.0];
      LAR1;
      L     LD 6;
      L     LD 2;
      R      [AR1,P#6.1];
      AN    #Eingang2;
      BLD   5;
      T     LD 2;
      TAK;
      T     LD 6;
      L     P##Zahler;
      LAR1;
      L     W [AR1,P#0.0];
      T     LW 0;
      OPN   DB [LW 0];
      L     D [AR1,P#2.0];
      LAR1;
      L     LD 6;
      L     LD 2;
      R      [AR1,P#6.2];
      BLD   5;
      T     LD 2;
      TAK;
      T     LD 6;
      L     P##Zahler;
      LAR1;
      L     W [AR1,P#0.0];
      T     LW 0;
      OPN   DB [LW 0];
      L     D [AR1,P#2.0];
      LAR1;
      L     LD 6;
      L     LD 2;
      R      [AR1,P#6.3];
      A     #Eingang1;
      BLD   5;
      T     LD 2;
      TAK;
      T     LD 6;
      L     P##Zahler;
      LAR1;
      L     W [AR1,P#0.0];
      T     LW 0;
      OPN   DB [LW 0];
      L     D [AR1,P#2.0];
      LAR1;
      L     LD 6;
      L     LD 2;
      AN     [AR1,P#6.0];
      BLD   5;
      T     LD 2;
      TAK;
      T     LD 6;
      L     P##Zahler;
      LAR1;
      L     W [AR1,P#0.0];
      T     LW 0;
      OPN   DB [LW 0];
      L     D [AR1,P#2.0];
      LAR1;
      L     LD 6;
      L     LD 2;
      S      [AR1,P#6.0];
      BLD   5;
      T     LD 2;
      TAK;
      T     LD 6;
      L     P##Zahler;
      LAR1;
      L     W [AR1,P#0.0];
      T     LW 0;
      OPN   DB [LW 0];
      L     D [AR1,P#2.0];
      LAR1;
      L     LD 6;
      L     LD 2;
      =      [AR1,P#6.1];
      A     #Eingang2;
      BLD   5;
      T     LD 2;
      TAK;
      T     LD 6;
      L     P##Zahler;
      LAR1;
      L     W [AR1,P#0.0];
      T     LW 0;
      OPN   DB [LW 0];
      L     D [AR1,P#2.0];
      LAR1;
      L     LD 6;
      L     LD 2;
      AN     [AR1,P#6.2];
      BLD   5;
      T     LD 2;
      TAK;
      T     LD 6;
      L     P##Zahler;
      LAR1;
      L     W [AR1,P#0.0];
      T     LW 0;
      OPN   DB [LW 0];
      L     D [AR1,P#2.0];
      LAR1;
      L     LD 6;
      L     LD 2;
      S      [AR1,P#6.2];
      BLD   5;
      T     LD 2;
      TAK;
      T     LD 6;
      L     P##Zahler;
      LAR1;
      L     W [AR1,P#0.0];
      T     LW 0;
      OPN   DB [LW 0];
      L     D [AR1,P#2.0];
      LAR1;
      L     LD 6;
      L     LD 2;
      =      [AR1,P#6.3];
NETWORK
TITLE = Counter device
      A     #Eingang1;	// Track A
      BLD   5;	// Track A pos Flanke
      T     LD 2;	// Track B pos Flanke
      TAK;
      T     LD 6;
      L     P##Zahler;
      LAR1;
      L     W [AR1,P#0.0];
      T     LW 0;
      OPN   DB [LW 0];	// Track B pos Flanke
      L     D [AR1,P#2.0];
      LAR1;	// Track B
      L     LD 6;	// Track B pos Flanke
      L     LD 2;	// Track A pos Flanke
      AN     [AR1,P#6.1];
      BLD   5;
      T     LD 2;
      TAK;
      T     LD 6;
      L     P##Zahler;
      LAR1;	// Track A pos Flanke
      L     W [AR1,P#0.0];
      T     LW 0;
      OPN   DB [LW 0];
      L     D [AR1,P#2.0];
      LAR1;
      L     LD 6;
      L     LD 2;
      A      [AR1,P#6.3];
      JCN   en05;
      BLD   5;
      T     LD 2;
      TAK;
      T     LD 6;
      L     P##Zahler;
      LAR1;
      L     W [AR1,P#0.0];
      T     LW 0;
      OPN   DB [LW 0];
      L     D [AR1,P#2.0];
      LAR1;
      L     LD 6;
      L     LD 2;
      L     D [AR1,P#8.0];
      L     1;
      +D;
      BLD   5;
      T     LD 2;
      TAK;
      T     LD 6;
      L     P##Zahler;
      LAR1;
      L     W [AR1,P#0.0];
      T     LW 0;
      OPN   DB [LW 0];
      L     D [AR1,P#2.0];
      LAR1;
      L     LD 6;
      L     LD 2;
      T     D [AR1,P#8.0];
      SET;
      BLD   5;
      T     LD 2;
      TAK;
      T     LD 6;
      L     P##Zahler;
      LAR1;
      L     W [AR1,P#0.0];
      T     LW 0;
      OPN   DB [LW 0];
      L     D [AR1,P#2.0];
      LAR1;
      L     LD 6;
      L     LD 2;
      R      [AR1,P#6.3];
en05: NOP   0;
      A     #Eingang2;
      BLD   5;
      T     LD 2;
      TAK;
      T     LD 6;
      L     P##Zahler;
      LAR1;
      L     W [AR1,P#0.0];
      T     LW 0;
      OPN   DB [LW 0];
      L     D [AR1,P#2.0];
      LAR1;
      L     LD 6;
      L     LD 2;
      AN     [AR1,P#6.3];
      BLD   5;
      T     LD 2;
      TAK;
      T     LD 6;
      L     P##Zahler;
      LAR1;
      L     W [AR1,P#0.0];
      T     LW 0;
      OPN   DB [LW 0];
      L     D [AR1,P#2.0];
      LAR1;
      L     LD 6;
      L     LD 2;
      A      [AR1,P#6.1];
      JCN   en06;
      BLD   5;
      T     LD 2;
      TAK;
      T     LD 6;
      L     P##Zahler;
      LAR1;
      L     W [AR1,P#0.0];
      T     LW 0;
      OPN   DB [LW 0];
      L     D [AR1,P#2.0];
      LAR1;
      L     LD 6;
      L     LD 2;
      L     D [AR1,P#8.0];
      L     1;
      -D;
      BLD   5;
      T     LD 2;
      TAK;
      T     LD 6;
      L     P##Zahler;
      LAR1;
      L     W [AR1,P#0.0];
      T     LW 0;
      OPN   DB [LW 0];
      L     D [AR1,P#2.0];
      LAR1;
      L     LD 6;
      L     LD 2;
      T     D [AR1,P#8.0];
      SET;
      BLD   5;
      T     LD 2;
      TAK;
      T     LD 6;
      L     P##Zahler;
      LAR1;
      L     W [AR1,P#0.0];
      T     LW 0;
      OPN   DB [LW 0];
      L     D [AR1,P#2.0];
      LAR1;
      L     LD 6;
      L     LD 2;
      R      [AR1,P#6.1];
en06: NOP   0;
END_FUNCTION

